screen "Lavados_Actuales" 1366x768, template "Pulsadores"
   Button "Botón_1" at 11,49 size 65x65; TextOff '1'
      on Click: SetTag("Ver_Anim_Boton", 1); SetTag("Ver_IDList", 0); "S400_ActListLav"(1)
      Appearance <- "Ver_Anim_Boton"
   IOField "Campo ES_1" at 115,75 size 95x32; FormatPattern 9999999999999999999999999999999999999999
      ProcessValue <- "Ver_HoraInicio_0"
   IOField "Campo ES_2" at 212,75 size 95x32; FormatPattern 9999999999999999999999999999999999999999
      ProcessValue <- "Ver_HoraFin_0"
   IOField "Campo ES_3" at 711,75 size 95x32; FormatPattern 99999
      ProcessValue <- "Ver_Carga_0"
   IOField "Campo ES_4" at 808,75 size 95x32; FormatPattern 99
      ProcessValue <- "Ver_Programa_0"
   IOField "Campo ES_5" at 309,75 size 400x32; FormatPattern ????????????????????????????????????????????????????????????????
      ProcessValue <- "Ver_Cli_Str_0"
   IOField "Campo ES_6" at 905,75 size 192x32; FormatPattern ????????????????????????????????????????????????????????????????
      ProcessValue <- "Ver_Operador_Str_0"
   IOField "Campo ES_7" at 115,106 size 95x32; FormatPattern 9999999999999999999999999999999999999999
      ProcessValue <- "Ver_HoraInicio_1"
   IOField "Campo ES_8" at 212,106 size 95x32; FormatPattern 9999999999999999999999999999999999999999
      ProcessValue <- "Ver_HoraFin_1"
   IOField "Campo ES_9" at 711,106 size 95x32; FormatPattern 99999
      ProcessValue <- "Ver_Carga_1"
   IOField "Campo ES_10" at 808,106 size 95x32; FormatPattern 99
      ProcessValue <- "Ver_Programa_1"
   IOField "Campo ES_11" at 309,106 size 400x32; FormatPattern ????????????????????????????????????????????????????????????????
      ProcessValue <- "Ver_Cli_Str_1"
   IOField "Campo ES_12" at 905,106 size 192x32; FormatPattern ????????????????????????????????????????????????????????????????
      ProcessValue <- "Ver_Operador_Str_1"
   IOField "Campo ES_13" at 115,137 size 95x32; FormatPattern 9999999999999999999999999999999999999999
      ProcessValue <- "Ver_HoraInicio_2"
   IOField "Campo ES_14" at 212,137 size 95x32; FormatPattern 9999999999999999999999999999999999999999
      ProcessValue <- "Ver_HoraFin_2"
   IOField "Campo ES_15" at 711,137 size 95x32; FormatPattern 99999
      ProcessValue <- "Ver_Carga_2"
   IOField "Campo ES_16" at 808,137 size 95x32; FormatPattern 99
      ProcessValue <- "Ver_Programa_2"
   IOField "Campo ES_17" at 309,137 size 400x32; FormatPattern ????????????????????????????????????????????????????????????????
      ProcessValue <- "Ver_Cli_Str_2"
   IOField "Campo ES_18" at 905,137 size 192x32; FormatPattern ????????????????????????????????????????????????????????????????
      ProcessValue <- "Ver_Operador_Str_2"
   IOField "Campo ES_19" at 115,168 size 95x32; FormatPattern 9999999999999999999999999999999999999999
      ProcessValue <- "Ver_HoraInicio_3"
   IOField "Campo ES_20" at 212,168 size 95x32; FormatPattern 9999999999999999999999999999999999999999
      ProcessValue <- "Ver_HoraFin_3"
   IOField "Campo ES_21" at 711,168 size 95x32; FormatPattern 99999
      ProcessValue <- "Ver_Carga_3"
   IOField "Campo ES_22" at 808,168 size 95x32; FormatPattern 99
      ProcessValue <- "Ver_Programa_3"
   IOField "Campo ES_23" at 309,168 size 400x32; FormatPattern ????????????????????????????????????????????????????????????????
      ProcessValue <- "Ver_Cli_Str_3"
   IOField "Campo ES_24" at 905,168 size 192x32; FormatPattern ????????????????????????????????????????????????????????????????
      ProcessValue <- "Ver_Operador_Str_3"
   IOField "Campo ES_25" at 115,199 size 95x32; FormatPattern 9999999999999999999999999999999999999999
      ProcessValue <- "Ver_HoraInicio_4"
   IOField "Campo ES_26" at 212,199 size 95x32; FormatPattern 9999999999999999999999999999999999999999
      ProcessValue <- "Ver_HoraFin_4"
   IOField "Campo ES_27" at 711,199 size 95x32; FormatPattern 99999
      ProcessValue <- "Ver_Carga_4"
   IOField "Campo ES_28" at 808,199 size 95x32; FormatPattern 99
      ProcessValue <- "Ver_Programa_4"
   IOField "Campo ES_29" at 309,199 size 400x32; FormatPattern ????????????????????????????????????????????????????????????????
      ProcessValue <- "Ver_Cli_Str_4"
   IOField "Campo ES_30" at 905,199 size 192x32; FormatPattern ????????????????????????????????????????????????????????????????
      ProcessValue <- "Ver_Operador_Str_4"
   IOField "Campo ES_31" at 115,230 size 95x32; FormatPattern 9999999999999999999999999999999999999999
      ProcessValue <- "Ver_HoraInicio_5"
   IOField "Campo ES_32" at 212,230 size 95x32; FormatPattern 9999999999999999999999999999999999999999
      ProcessValue <- "Ver_HoraFin_5"
   IOField "Campo ES_33" at 711,230 size 95x32; FormatPattern 99999
      ProcessValue <- "Ver_Carga_5"
   IOField "Campo ES_34" at 808,230 size 95x32; FormatPattern 99
      ProcessValue <- "Ver_Programa_5"
   IOField "Campo ES_35" at 309,230 size 400x32; FormatPattern ????????????????????????????????????????????????????????????????
      ProcessValue <- "Ver_Cli_Str_5"
   IOField "Campo ES_36" at 905,230 size 192x32; FormatPattern ????????????????????????????????????????????????????????????????
      ProcessValue <- "Ver_Operador_Str_5"
   IOField "Campo ES_37" at 115,261 size 95x32; FormatPattern 9999999999999999999999999999999999999999
      ProcessValue <- "Ver_HoraInicio_6"
   IOField "Campo ES_38" at 212,261 size 95x32; FormatPattern 9999999999999999999999999999999999999999
      ProcessValue <- "Ver_HoraFin_6"
   IOField "Campo ES_39" at 711,261 size 95x32; FormatPattern 99999
      ProcessValue <- "Ver_Carga_6"
   IOField "Campo ES_40" at 808,261 size 95x32; FormatPattern 99
      ProcessValue <- "Ver_Programa_6"
   IOField "Campo ES_41" at 309,261 size 400x32; FormatPattern ????????????????????????????????????????????????????????????????
      ProcessValue <- "Ver_Cli_Str_6"
   IOField "Campo ES_42" at 905,261 size 192x32; FormatPattern ????????????????????????????????????????????????????????????????
      ProcessValue <- "Ver_Operador_Str_6"
   IOField "Campo ES_43" at 115,292 size 95x32; FormatPattern 9999999999999999999999999999999999999999
      ProcessValue <- "Ver_HoraInicio_7"
   IOField "Campo ES_44" at 212,292 size 95x32; FormatPattern 9999999999999999999999999999999999999999
      ProcessValue <- "Ver_HoraFin_7"
   IOField "Campo ES_45" at 711,292 size 95x32; FormatPattern 99999
      ProcessValue <- "Ver_Carga_7"
   IOField "Campo ES_46" at 808,292 size 95x32; FormatPattern 99
      ProcessValue <- "Ver_Programa_7"
   IOField "Campo ES_47" at 309,292 size 400x32; FormatPattern ????????????????????????????????????????????????????????????????
      ProcessValue <- "Ver_Cli_Str_7"
   IOField "Campo ES_48" at 905,292 size 192x32; FormatPattern ????????????????????????????????????????????????????????????????
      ProcessValue <- "Ver_Operador_Str_7"
   IOField "Campo ES_49" at 115,323 size 95x32; FormatPattern 9999999999999999999999999999999999999999
      ProcessValue <- "Ver_HoraInicio_8"
   IOField "Campo ES_50" at 212,323 size 95x32; FormatPattern 9999999999999999999999999999999999999999
      ProcessValue <- "Ver_HoraFin_8"
   IOField "Campo ES_51" at 711,323 size 95x32; FormatPattern 99999
      ProcessValue <- "Ver_Carga_8"
   IOField "Campo ES_52" at 808,323 size 95x32; FormatPattern 99
      ProcessValue <- "Ver_Programa_8"
   IOField "Campo ES_53" at 309,323 size 400x32; FormatPattern ????????????????????????????????????????????????????????????????
      ProcessValue <- "Ver_Cli_Str_8"
   IOField "Campo ES_54" at 905,323 size 192x32; FormatPattern ????????????????????????????????????????????????????????????????
      ProcessValue <- "Ver_Operador_Str_8"
   IOField "Campo ES_55" at 115,354 size 95x32; FormatPattern 9999999999999999999999999999999999999999
      ProcessValue <- "Ver_HoraInicio_9"
   IOField "Campo ES_56" at 212,354 size 95x32; FormatPattern 9999999999999999999999999999999999999999
      ProcessValue <- "Ver_HoraFin_9"
   IOField "Campo ES_57" at 711,354 size 95x32; FormatPattern 99999
      ProcessValue <- "Ver_Carga_9"
   IOField "Campo ES_58" at 808,354 size 95x32; FormatPattern 99
      ProcessValue <- "Ver_Programa_9"
   IOField "Campo ES_59" at 309,354 size 400x32; FormatPattern ????????????????????????????????????????????????????????????????
      ProcessValue <- "Ver_Cli_Str_9"
   IOField "Campo ES_60" at 905,354 size 192x32; FormatPattern ????????????????????????????????????????????????????????????????
      ProcessValue <- "Ver_Operador_Str_9"
   IOField "Campo ES_61" at 115,385 size 95x32; FormatPattern 9999999999999999999999999999999999999999
      ProcessValue <- "Ver_HoraInicio_10"
   IOField "Campo ES_62" at 212,385 size 95x32; FormatPattern 9999999999999999999999999999999999999999
      ProcessValue <- "Ver_HoraFin_10"
   IOField "Campo ES_63" at 711,385 size 95x32; FormatPattern 99999
      ProcessValue <- "Ver_Carga_10"
   IOField "Campo ES_64" at 808,385 size 95x32; FormatPattern 99
      ProcessValue <- "Ver_Programa_10"
   IOField "Campo ES_65" at 309,385 size 400x32; FormatPattern ????????????????????????????????????????????????????????????????
      ProcessValue <- "Ver_Cli_Str_10"
   IOField "Campo ES_66" at 905,385 size 192x32; FormatPattern ????????????????????????????????????????????????????????????????
      ProcessValue <- "Ver_Operador_Str_10"
   IOField "Campo ES_67" at 115,416 size 95x32; FormatPattern 9999999999999999999999999999999999999999
      ProcessValue <- "Ver_HoraInicio_11"
   IOField "Campo ES_68" at 212,416 size 95x32; FormatPattern 9999999999999999999999999999999999999999
      ProcessValue <- "Ver_HoraFin_11"
   IOField "Campo ES_69" at 711,416 size 95x32; FormatPattern 99999
      ProcessValue <- "Ver_Carga_11"
   IOField "Campo ES_70" at 808,416 size 95x32; FormatPattern 99
      ProcessValue <- "Ver_Programa_11"
   IOField "Campo ES_71" at 309,416 size 400x32; FormatPattern ????????????????????????????????????????????????????????????????
      ProcessValue <- "Ver_Cli_Str_11"
   IOField "Campo ES_72" at 905,416 size 192x32; FormatPattern ????????????????????????????????????????????????????????????????
      ProcessValue <- "Ver_Operador_Str_11"
   IOField "Campo ES_73" at 115,447 size 95x32; FormatPattern 9999999999999999999999999999999999999999
      ProcessValue <- "Ver_HoraInicio_12"
   IOField "Campo ES_74" at 212,447 size 95x32; FormatPattern 9999999999999999999999999999999999999999
      ProcessValue <- "Ver_HoraFin_12"
   IOField "Campo ES_75" at 711,447 size 95x32; FormatPattern 99999
      ProcessValue <- "Ver_Carga_12"
   IOField "Campo ES_76" at 808,447 size 95x32; FormatPattern 99
      ProcessValue <- "Ver_Programa_12"
   IOField "Campo ES_77" at 309,447 size 400x32; FormatPattern ????????????????????????????????????????????????????????????????
      ProcessValue <- "Ver_Cli_Str_12"
   IOField "Campo ES_78" at 905,447 size 192x32; FormatPattern ????????????????????????????????????????????????????????????????
      ProcessValue <- "Ver_Operador_Str_12"
   IOField "Campo ES_79" at 115,478 size 95x32; FormatPattern 9999999999999999999999999999999999999999
      ProcessValue <- "Ver_HoraInicio_13"
   IOField "Campo ES_80" at 212,478 size 95x32; FormatPattern 9999999999999999999999999999999999999999
      ProcessValue <- "Ver_HoraFin_13"
   IOField "Campo ES_81" at 711,478 size 95x32; FormatPattern 99999
      ProcessValue <- "Ver_Carga_13"
   IOField "Campo ES_82" at 808,478 size 95x32; FormatPattern 99
      ProcessValue <- "Ver_Programa_13"
   IOField "Campo ES_83" at 309,478 size 400x32; FormatPattern ????????????????????????????????????????????????????????????????
      ProcessValue <- "Ver_Cli_Str_13"
   IOField "Campo ES_84" at 905,478 size 192x32; FormatPattern ????????????????????????????????????????????????????????????????
      ProcessValue <- "Ver_Operador_Str_13"
   IOField "Campo ES_85" at 115,509 size 95x32; FormatPattern 9999999999999999999999999999999999999999
      ProcessValue <- "Ver_HoraInicio_14"
   IOField "Campo ES_86" at 212,509 size 95x32; FormatPattern 9999999999999999999999999999999999999999
      ProcessValue <- "Ver_HoraFin_14"
   IOField "Campo ES_87" at 711,509 size 95x32; FormatPattern 99999
      ProcessValue <- "Ver_Carga_14"
   IOField "Campo ES_88" at 808,509 size 95x32; FormatPattern 99
      ProcessValue <- "Ver_Programa_14"
   IOField "Campo ES_89" at 309,509 size 400x32; FormatPattern ????????????????????????????????????????????????????????????????
      ProcessValue <- "Ver_Cli_Str_14"
   IOField "Campo ES_90" at 905,509 size 192x32; FormatPattern ????????????????????????????????????????????????????????????????
      ProcessValue <- "Ver_Operador_Str_14"
   TextField "Campo de texto_1" at 115,41 size 95x32; Text 'INICIO'
   TextField "Campo de texto_2" at 212,41 size 95x32; Text 'FIN'
   TextField "Campo de texto_3" at 309,41 size 95x32; Text 'CLIENTES'
   TextField "Campo de texto_4" at 711,41 size 95x32; Text 'CARGA'
   TextField "Campo de texto_5" at 808,41 size 95x32; Text 'PROG'
   TextField "Campo de texto_6" at 913,41 size 95x32; Text 'OPERADOR'
   Button "Botón_3" at 1145,665 size 39x38; TextOff 'Text'
      on Click: function_b9b71300("Ver_IDList", 1); "S400_ActListLav"("Ver_Anim_Boton")
   Button "Botón_4" at 1145,41 size 39x38; TextOff 'Text'
      on Click: function_dd21b452("Ver_IDList", 1); "S400_ActListLav"("Ver_Anim_Boton")
   Button "Botón_5" at 10,126 size 65x65; TextOff '2'
      on Click: SetTag("Ver_IDList", 0); SetTag("Ver_Anim_Boton", 2); "S400_ActListLav"(2)
      Appearance <- "Ver_Anim_Boton"
   Button "Botón_6" at 10,205 size 65x65; TextOff '3'
      on Click: SetTag("Ver_IDList", 0); SetTag("Ver_Anim_Boton", 3); "S400_ActListLav"(3)
      Appearance <- "Ver_Anim_Boton"
   Button "Botón_7" at 10,284 size 65x65; TextOff '4'
      on Click: SetTag("Ver_IDList", 0); SetTag("Ver_Anim_Boton", 4); "S400_ActListLav"(4)
      Appearance <- "Ver_Anim_Boton"
   IOField "Campo ES_91" at 115,541 size 95x32; FormatPattern 9999999999999999999999999999999999999999
      ProcessValue <- "Ver_HoraInicio_14"
   IOField "Campo ES_92" at 212,541 size 95x32; FormatPattern 9999999999999999999999999999999999999999
      ProcessValue <- "Ver_HoraFin_14"
   IOField "Campo ES_93" at 711,541 size 95x32; FormatPattern 99999
      ProcessValue <- "Ver_Carga_14"
   IOField "Campo ES_94" at 808,541 size 95x32; FormatPattern 99
      ProcessValue <- "Ver_Programa_14"
   IOField "Campo ES_95" at 309,541 size 400x32; FormatPattern ????????????????????????????????????????????????????????????????
      ProcessValue <- "Ver_Cli_Str_14"
   IOField "Campo ES_96" at 905,541 size 192x32; FormatPattern ????????????????????????????????????????????????????????????????
      ProcessValue <- "Ver_Operador_Str_14"
   IOField "Campo ES_97" at 115,573 size 95x32; FormatPattern 9999999999999999999999999999999999999999
      ProcessValue <- "Ver_HoraInicio_14"
   IOField "Campo ES_98" at 212,573 size 95x32; FormatPattern 9999999999999999999999999999999999999999
      ProcessValue <- "Ver_HoraFin_14"
   IOField "Campo ES_99" at 711,573 size 95x32; FormatPattern 99999
      ProcessValue <- "Ver_Carga_14"
   IOField "Campo ES_100" at 808,573 size 95x32; FormatPattern 99
      ProcessValue <- "Ver_Programa_14"
   IOField "Campo ES_101" at 309,573 size 400x32; FormatPattern ????????????????????????????????????????????????????????????????
      ProcessValue <- "Ver_Cli_Str_14"
   IOField "Campo ES_102" at 905,573 size 192x32; FormatPattern ????????????????????????????????????????????????????????????????
      ProcessValue <- "Ver_Operador_Str_14"
   IOField "Campo ES_103" at 115,605 size 95x32; FormatPattern 9999999999999999999999999999999999999999
      ProcessValue <- "Ver_HoraInicio_14"
   IOField "Campo ES_104" at 212,605 size 95x32; FormatPattern 9999999999999999999999999999999999999999
      ProcessValue <- "Ver_HoraFin_14"
   IOField "Campo ES_105" at 711,605 size 95x32; FormatPattern 99999
      ProcessValue <- "Ver_Carga_14"
   IOField "Campo ES_106" at 808,605 size 95x32; FormatPattern 99
      ProcessValue <- "Ver_Programa_14"
   IOField "Campo ES_107" at 309,605 size 400x32; FormatPattern ????????????????????????????????????????????????????????????????
      ProcessValue <- "Ver_Cli_Str_14"
   IOField "Campo ES_108" at 905,605 size 192x32; FormatPattern ????????????????????????????????????????????????????????????????
      ProcessValue <- "Ver_Operador_Str_14"
   IOField "Campo ES_109" at 115,637 size 95x32; FormatPattern 9999999999999999999999999999999999999999
      ProcessValue <- "Ver_HoraInicio_14"
   IOField "Campo ES_110" at 212,637 size 95x32; FormatPattern 9999999999999999999999999999999999999999
      ProcessValue <- "Ver_HoraFin_14"
   IOField "Campo ES_111" at 711,637 size 95x32; FormatPattern 99999
      ProcessValue <- "Ver_Carga_14"
   IOField "Campo ES_112" at 808,637 size 95x32; FormatPattern 99
      ProcessValue <- "Ver_Programa_14"
   IOField "Campo ES_113" at 309,637 size 400x32; FormatPattern ????????????????????????????????????????????????????????????????
      ProcessValue <- "Ver_Cli_Str_14"
   IOField "Campo ES_114" at 905,637 size 192x32; FormatPattern ????????????????????????????????????????????????????????????????
      ProcessValue <- "Ver_Operador_Str_14"
   IOField "Campo ES_115" at 115,669 size 95x32; FormatPattern 9999999999999999999999999999999999999999
      ProcessValue <- "Ver_HoraInicio_14"
   IOField "Campo ES_116" at 212,669 size 95x32; FormatPattern 9999999999999999999999999999999999999999
      ProcessValue <- "Ver_HoraFin_14"
   IOField "Campo ES_117" at 711,669 size 95x32; FormatPattern 99999
      ProcessValue <- "Ver_Carga_14"
   IOField "Campo ES_118" at 808,669 size 95x32; FormatPattern 99
      ProcessValue <- "Ver_Programa_14"
   IOField "Campo ES_119" at 309,669 size 400x32; FormatPattern ????????????????????????????????????????????????????????????????
      ProcessValue <- "Ver_Cli_Str_14"
   IOField "Campo ES_120" at 905,669 size 192x32; FormatPattern ????????????????????????????????????????????????????????????????
      ProcessValue <- "Ver_Operador_Str_14"
   TextField "Campo de texto_7" at 1099,75 size 32x32; Text 'X'
   TextField "Campo de texto_8" at 1099,106 size 32x32; Text 'X'
   TextField "Campo de texto_9" at 1099,137 size 32x32; Text 'X'
   TextField "Campo de texto_10" at 1099,168 size 32x32; Text 'X'
   TextField "Campo de texto_11" at 1099,199 size 32x32; Text 'X'
   TextField "Campo de texto_12" at 1099,230 size 32x32; Text 'X'
   TextField "Campo de texto_13" at 1099,261 size 32x32; Text 'X'
   TextField "Campo de texto_14" at 1099,292 size 32x32; Text 'X'
   TextField "Campo de texto_15" at 1099,323 size 32x32; Text 'X'
   TextField "Campo de texto_16" at 1099,354 size 32x32; Text 'X'
   TextField "Campo de texto_17" at 1099,385 size 32x32; Text 'X'
   TextField "Campo de texto_18" at 1099,416 size 32x32; Text 'X'
   TextField "Campo de texto_19" at 1099,447 size 32x32; Text 'X'
   TextField "Campo de texto_20" at 1099,478 size 32x32; Text 'X'
   TextField "Campo de texto_21" at 1099,509 size 32x32; Text 'X'
   TextField "Campo de texto_22" at 1099,541 size 32x32; Text 'X'
   TextField "Campo de texto_23" at 1099,573 size 32x32; Text 'X'
   TextField "Campo de texto_24" at 1099,605 size 32x32; Text 'X'
   TextField "Campo de texto_25" at 1099,637 size 32x32; Text 'X'
   TextField "Campo de texto_26" at 1099,669 size 32x32; Text 'X'
   Group "Group" at 1099,75 size 32x32
   Group "Group_1" at 1099,106 size 32x32
   Group "Group_2" at 1099,137 size 32x32
   Group "Group_3" at 1099,168 size 32x32
   Group "Group_4" at 1099,199 size 32x32
   Group "Group_5" at 1099,230 size 32x32
   Group "Group_6" at 1099,261 size 32x32
   Group "Group_7" at 1099,292 size 32x32
   Group "Group_8" at 1099,323 size 32x32
   Group "Group_9" at 1099,354 size 32x32
   Group "Group_10" at 1099,385 size 32x32
   Group "Group_11" at 1099,416 size 32x32
   Group "Group_12" at 1099,447 size 32x32
   Group "Group_13" at 1099,478 size 32x32
   Group "Group_14" at 1099,509 size 32x32
   Group "Group_15" at 1099,541 size 32x32
   Group "Group_16" at 1099,573 size 32x32
   Group "Group_17" at 1099,605 size 32x32
   Group "Group_18" at 1099,637 size 32x32
   Group "Group_19" at 1099,669 size 32x32
   Button "Botón_8" at 1200,75 size 32x32; TextOff 'E'
      Visibility <- "Ver_Programa_0"
      on Click: SetBit("Ver_Editor_X"); "S402_ActRegDeEdicion"("Ver_Anim_Boton", 0)
   Button "Botón_11" at 13,6 size 65x32; TextOff 'HOY'
      on Click: "S403_ActDia"()
   IOField "Campo ES_133" at 101,6 size 115x32; FormatPattern 9999999999999999999999999999999999999999
      ProcessValue <- "Ver_DIA_X"
   Button "Botón_13" at 1200,106 size 32x32; TextOff 'E'
      on Click: SetBit("Ver_Editor_X"); "S402_ActRegDeEdicion"("Ver_Anim_Boton", 1)
      Visibility <- "Ver_Programa_1"
   Button "Botón_14" at 1200,137 size 32x32; TextOff 'E'
      on Click: SetBit("Ver_Editor_X"); "S402_ActRegDeEdicion"("Ver_Anim_Boton", 2)
      Visibility <- "Ver_Programa_2"
   Button "Botón_15" at 1200,168 size 32x32; TextOff 'E'
      on Click: SetBit("Ver_Editor_X"); "S402_ActRegDeEdicion"("Ver_Anim_Boton", 3)
      Visibility <- "Ver_Programa_3"
   Button "Botón_16" at 1200,199 size 32x32; TextOff 'E'
      on Click: SetBit("Ver_Editor_X"); "S402_ActRegDeEdicion"("Ver_Anim_Boton", 4)
      Visibility <- "Ver_Programa_4"
   Button "Botón_17" at 1200,230 size 32x32; TextOff 'E'
      on Click: SetBit("Ver_Editor_X"); "S402_ActRegDeEdicion"("Ver_Anim_Boton", 5)
      Visibility <- "Ver_Programa_5"
   Button "Botón_18" at 1200,261 size 32x32; TextOff 'E'
      on Click: SetBit("Ver_Editor_X"); "S402_ActRegDeEdicion"("Ver_Anim_Boton", 6)
      Visibility <- "Ver_Programa_6"
   Button "Botón_19" at 1200,292 size 32x32; TextOff 'E'
      on Click: SetBit("Ver_Editor_X"); "S402_ActRegDeEdicion"("Ver_Anim_Boton", 7)
      Visibility <- "Ver_Programa_7"
   Button "Botón_20" at 1200,323 size 32x32; TextOff 'E'
      on Click: SetBit("Ver_Editor_X"); "S402_ActRegDeEdicion"("Ver_Anim_Boton", 8)
      Visibility <- "Ver_Programa_8"
   Button "Botón_21" at 1200,354 size 32x32; TextOff 'E'
      on Click: SetBit("Ver_Editor_X"); "S402_ActRegDeEdicion"("Ver_Anim_Boton", 9)
      Visibility <- "Ver_Programa_9"
   Button "Botón_22" at 1200,385 size 32x32; TextOff 'E'
      on Click: SetBit("Ver_Editor_X"); "S402_ActRegDeEdicion"("Ver_Anim_Boton", 10)
      Visibility <- "Ver_Programa_10"
   Button "Botón_23" at 1200,416 size 32x32; TextOff 'E'
      on Click: SetBit("Ver_Editor_X"); "S402_ActRegDeEdicion"("Ver_Anim_Boton", 11)
      Visibility <- "Ver_Programa_11"
   Button "Botón_24" at 1200,447 size 32x32; TextOff 'E'
      on Click: SetBit("Ver_Editor_X"); "S402_ActRegDeEdicion"("Ver_Anim_Boton", 12)
      Visibility <- "Ver_Programa_12"
   Button "Botón_25" at 1200,478 size 32x32; TextOff 'E'
      on Click: SetBit("Ver_Editor_X"); "S402_ActRegDeEdicion"("Ver_Anim_Boton", 13)
      Visibility <- "Ver_Programa_13"
   Button "Botón_26" at 1200,509 size 32x32; TextOff 'E'
      on Click: SetBit("Ver_Editor_X"); "S402_ActRegDeEdicion"("Ver_Anim_Boton", 14)
      Visibility <- "Ver_Programa_14"
   Button "Botón_27" at 1200,541 size 32x32; TextOff 'E'
      on Click: SetBit("Ver_Editor_X"); "S402_ActRegDeEdicion"("Ver_Anim_Boton", 15)
      Visibility <- "Ver_Programa_15"
   Button "Botón_29" at 1200,573 size 32x32; TextOff 'E'
      on Click: SetBit("Ver_Editor_X"); "S402_ActRegDeEdicion"("Ver_Anim_Boton", 16)
      Visibility <- "Ver_Programa_16"
   Button "Botón_30" at 1200,605 size 32x32; TextOff 'E'
      on Click: SetBit("Ver_Editor_X"); "S402_ActRegDeEdicion"("Ver_Anim_Boton", 17)
      Visibility <- "Ver_Programa_17"
   Button "Botón_31" at 1200,637 size 32x32; TextOff 'E'
      on Click: SetBit("Ver_Editor_X"); "S402_ActRegDeEdicion"("Ver_Anim_Boton", 18)
      Visibility <- "Ver_Programa_18"
   Button "Botón_32" at 1200,669 size 32x32; TextOff 'E'
      on Click: SetBit("Ver_Editor_X"); "S402_ActRegDeEdicion"("Ver_Anim_Boton", 19)
      Visibility <- "Ver_Programa_19"
   Button "Botón_2" at 1045,720 size 161x48; TextOff 'PRINCIPAL'
      on Click: ActivateScreen("Principal", 0)
   Button "Botón_12" at 405,720 size 161x48; TextOff 'GENERAR INFORME'
      on Click: "S23_Creador_InformeDiarioLavs_Gral"(N)
   Rectangle "Rectángulo_2" at 1099,75 size 32x32
      Visibility <- "Ver_CicloValido_0"
   Polygon "Polígono_3" at 1103,78 size 23x24
      Visibility <- "Ver_CicloValido_0"
   Rectangle "Rectángulo_3" at 1099,106 size 32x32
      Visibility <- "Ver_CicloValido_1"
   Polygon "Polígono_4" at 1103,109 size 23x24
      Visibility <- "Ver_CicloValido_1"
   Rectangle "Rectángulo_4" at 1099,137 size 32x32
      Visibility <- "Ver_CicloValido_2"
   Polygon "Polígono_5" at 1103,140 size 23x24
      Visibility <- "Ver_CicloValido_2"
   Rectangle "Rectángulo_5" at 1099,168 size 32x32
      Visibility <- "Ver_CicloValido_3"
   Polygon "Polígono_6" at 1103,171 size 23x24
      Visibility <- "Ver_CicloValido_3"
   Rectangle "Rectángulo_6" at 1099,199 size 32x32
      Visibility <- "Ver_CicloValido_4"
   Polygon "Polígono_7" at 1103,202 size 23x24
      Visibility <- "Ver_CicloValido_4"
   Rectangle "Rectángulo_7" at 1099,230 size 32x32
      Visibility <- "Ver_CicloValido_5"
   Polygon "Polígono_8" at 1103,233 size 23x24
      Visibility <- "Ver_CicloValido_5"
   Rectangle "Rectángulo_8" at 1099,261 size 32x32
      Visibility <- "Ver_CicloValido_6"
   Polygon "Polígono_9" at 1103,264 size 23x24
      Visibility <- "Ver_CicloValido_6"
   Rectangle "Rectángulo_9" at 1099,292 size 32x32
      Visibility <- "Ver_CicloValido_7"
   Polygon "Polígono_10" at 1103,295 size 23x24
      Visibility <- "Ver_CicloValido_7"
   Rectangle "Rectángulo_10" at 1099,323 size 32x32
      Visibility <- "Ver_CicloValido_8"
   Polygon "Polígono_11" at 1103,326 size 23x24
      Visibility <- "Ver_CicloValido_8"
   Rectangle "Rectángulo_11" at 1099,354 size 32x32
      Visibility <- "Ver_CicloValido_9"
   Polygon "Polígono_12" at 1103,357 size 23x24
      Visibility <- "Ver_CicloValido_9"
   Rectangle "Rectángulo_12" at 1099,385 size 32x32
      Visibility <- "Ver_CicloValido_10"
   Polygon "Polígono_13" at 1103,388 size 23x24
      Visibility <- "Ver_CicloValido_10"
   Rectangle "Rectángulo_13" at 1099,416 size 32x32
      Visibility <- "Ver_CicloValido_11"
   Polygon "Polígono_14" at 1103,419 size 23x24
      Visibility <- "Ver_CicloValido_11"
   Rectangle "Rectángulo_14" at 1099,447 size 32x32
      Visibility <- "Ver_CicloValido_12"
   Polygon "Polígono_15" at 1103,450 size 23x24
      Visibility <- "Ver_CicloValido_12"
   Rectangle "Rectángulo_15" at 1099,478 size 32x32
      Visibility <- "Ver_CicloValido_13"
   Polygon "Polígono_16" at 1103,481 size 23x24
      Visibility <- "Ver_CicloValido_13"
   Rectangle "Rectángulo_16" at 1099,509 size 32x32
      Visibility <- "Ver_CicloValido_14"
   Polygon "Polígono_17" at 1103,512 size 23x24
      Visibility <- "Ver_CicloValido_14"
   Rectangle "Rectángulo_17" at 1099,541 size 32x32
      Visibility <- "Ver_CicloValido_15"
   Polygon "Polígono_18" at 1103,544 size 23x24
      Visibility <- "Ver_CicloValido_15"
   Rectangle "Rectángulo_18" at 1099,573 size 32x32
      Visibility <- "Ver_CicloValido_16"
   Polygon "Polígono_19" at 1103,576 size 23x24
      Visibility <- "Ver_CicloValido_16"
   Rectangle "Rectángulo_19" at 1099,605 size 32x32
      Visibility <- "Ver_CicloValido_17"
   Polygon "Polígono_20" at 1103,608 size 23x24
      Visibility <- "Ver_CicloValido_17"
   Rectangle "Rectángulo_20" at 1099,637 size 32x32
      Visibility <- "Ver_CicloValido_18"
   Polygon "Polígono_21" at 1103,640 size 23x24
      Visibility <- "Ver_CicloValido_18"
   Rectangle "Rectángulo_21" at 1099,669 size 32x32
      Visibility <- "Ver_CicloValido_19"
   Polygon "Polígono_22" at 1103,672 size 23x24
      Visibility <- "Ver_CicloValido_19"
   Rectangle "Rectángulo_22" at 101,250 size 1086x267
      Visibility <- "Ver_Editor_X"
   TextField "Campo de texto_33" at 134,265 size 185x16; Text 'REGISTRO ACTUAL'
      Visibility <- "Ver_Editor_X"
   TextField "Campo de texto_27" at 115,289 size 95x16; Text 'INICIO'
      Visibility <- "Ver_Editor_X"
   TextField "Campo de texto_28" at 212,289 size 95x16; Text 'FIN'
      Visibility <- "Ver_Editor_X"
   IOField "Campo ES_122" at 212,311 size 95x32; FormatPattern 9999999999999999999999999999999999999999
      Visibility <- "Ver_Editor_X"
      ProcessValue <- "Ver_HoraFin_X_ans"
   IOField "Campo ES_121" at 115,311 size 95x32; FormatPattern 9999999999999999999999999999999999999999
      Visibility <- "Ver_Editor_X"
      ProcessValue <- "Ver_HoraInicio_X_ans"
   TextField "Campo de texto_29" at 309,289 size 95x16; Text 'CLIENTES'
      Visibility <- "Ver_Editor_X"
   IOField "Campo ES_123" at 711,311 size 95x32; FormatPattern 99999
      Visibility <- "Ver_Editor_X"
      ProcessValue <- "Ver_Carga_X_ans"
   TextField "Campo de texto_30" at 711,289 size 95x16; Text 'CARGA'
      Visibility <- "Ver_Editor_X"
   TextField "Campo de texto_31" at 808,289 size 95x16; Text 'PROG'
      Visibility <- "Ver_Editor_X"
   IOField "Campo ES_124" at 808,311 size 95x32; FormatPattern 99
      Visibility <- "Ver_Editor_X"
      ProcessValue <- "Ver_Programa_X_ans"
   TextField "Campo de texto_32" at 913,289 size 95x16; Text 'OPERADOR'
      Visibility <- "Ver_Editor_X"
   TextField "Campo de texto_39" at 913,388 size 95x16; Text 'OPERADOR'
      Visibility <- "Ver_Editor_X"
   TextField "Campo de texto_38" at 808,388 size 95x16; Text 'PROG'
      Visibility <- "Ver_Editor_X"
   TextField "Campo de texto_37" at 711,388 size 95x16; Text 'CARGA'
      Visibility <- "Ver_Editor_X"
   TextField "Campo de texto_35" at 212,388 size 95x16; Text 'FIN'
      Visibility <- "Ver_Editor_X"
   TextField "Campo de texto_40" at 134,364 size 185x16; Text 'REGISTRO NUEVO'
      Visibility <- "Ver_Editor_X"
   TextField "Campo de texto_34" at 115,388 size 95x16; Text 'INICIO'
      Visibility <- "Ver_Editor_X"
   Button "Botón_9" at 893,455 size 132x34; TextOff 'Guardar'
      Visibility <- "Ver_Editor_X"
      on Click: "S401_EditarLavado"("Ver_Anim_Boton"); ResetBit("Ver_Editor_X")
   Button "Botón_10" at 1035,455 size 132x34; TextOff 'Cancelar'
      Visibility <- "Ver_Editor_X"
      on Click: SetTag("Ver_CicloValido_X", 0); ResetBit("Ver_Editor_X")
   SymbolicIOField "Campo ES simbólico_2" at 309,407 size 400x32; TextOff '0'; TextOn '1'; TextList "Clientes"
      ProcessValue <- "Ver_Cli1_Str_X"
      Visibility <- "Ver_Editor_X"
   SymbolicIOField "Campo ES simbólico_1" at 309,441 size 400x32; TextOn '1'; TextOff '0'; TextList "Clientes"
      Visibility <- "Ver_Editor_X"
      ProcessValue <- "Ver_Cli2_Str_X"
   SymbolicIOField "Campo ES simbólico_3" at 309,475 size 400x32; TextOn '1'; TextOff '0'; TextList "Clientes"
      Visibility <- "Ver_Editor_X"
      ProcessValue <- "Ver_Cli3_Str_X"
   SymbolicIOField "Campo ES simbólico_4" at 905,407 size 192x32; TextOn '1'; TextOff '0'; TextList "Operadores_Lavadora"
      ProcessValue <- "Ver_Operador_Int_X"
      Visibility <- "Ver_Editor_X"
   IOField "Campo ES_131" at 808,407 size 95x32; FormatPattern 99
      ProcessValue <- "Ver_Programa_X"
      Visibility <- "Ver_Editor_X"
   IOField "Campo ES_129" at 711,407 size 95x32; FormatPattern 99999
      ProcessValue <- "Ver_Carga_X"
      Visibility <- "Ver_Editor_X"
   IOField "Campo ES_130" at 115,407 size 95x32; FormatPattern 9999999999999999999999999999999999999999
      ProcessValue <- "Ver_HoraInicio_X"
      Visibility <- "Ver_Editor_X"
   IOField "Campo ES_127" at 212,407 size 95x32; FormatPattern 9999999999999999999999999999999999999999
      ProcessValue <- "Ver_HoraFin_X"
      Visibility <- "Ver_Editor_X"
   SymbolicIOField "Campo ES simbólico_5" at 309,311 size 400x24; TextOn '1'; TextOff '0'; TextList "Clientes"
      Visibility <- "Ver_Editor_X"
      ProcessValue <- "Ver_Cli1_Str_X_ans"
   SymbolicIOField "Campo ES simbólico_6" at 309,337 size 400x24; TextOn '1'; TextOff '0'; TextList "Clientes"
      Visibility <- "Ver_Editor_X"
      ProcessValue <- "Ver_Cli2_Str_X_ans"
   SymbolicIOField "Campo ES simbólico_7" at 309,363 size 400x24; TextOn '1'; TextOff '0'; TextList "Clientes"
      Visibility <- "Ver_Editor_X"
      ProcessValue <- "Ver_Cli3_Str_X_ans"
   SymbolicIOField "Campo ES simbólico_8" at 905,311 size 192x32; TextOn '1'; TextOff '0'; TextList "Operadores_Lavadora"
      Visibility <- "Ver_Editor_X"
      ProcessValue <- "Ver_Operador_Int_X_ans"
   Switch "Interruptor_1" at 1099,311 size 63x32; CaptionText 'Switch'; TextOff 'NO'; TextOn 'SI'
      ProcessValue <- "Ver_CicloValido_X_ans"
      Visibility <- "Ver_Editor_X"
   Switch "Interruptor_2" at 1099,407 size 63x32; TextOn 'SI'; CaptionText 'Switch'; TextOff 'NO'
      ProcessValue <- "Ver_CicloValido_X"
      Visibility <- "Ver_Editor_X"

screen "Informes" 1366x768, template "Pulsadores"
   Button "Botón_3" at 725,720 size 161x48; TextOff 'LAVADOS'
      on Click: ActivateScreen("Lavados_Actuales", 0); "S403_ActDia"()
   Button "Botón_8" at 1045,720 size 161x48; TextOff 'PRINCIPAL'
      on Click: ActivateScreen("Principal", 0)
   Button "Botón_1" at 414,456 size 161x48; TextOff 'GENERAR INFORME'
      on Click: "S500_InformePeriodico"(1, "Inf_Ano", "Inf_Mes")
   IOField "Campo ES_1" at 167,456 size 50x48; FormatPattern 99
      ProcessValue <- "Inf_Mes"
   IOField "Campo ES_2" at 161,130 size 170x48; FormatPattern 9999999999999999999999999999999999999999
      ProcessValue <- "Inf_Desde"
   IOField "Campo ES_3" at 161,194 size 170x48; FormatPattern 9999999999999999999999999999999999999999
      ProcessValue <- "Inf_Hasta"
   TextField "Campo de texto_1" at 86,464 size 55x32; Text 'MES'
   TextField "Campo de texto_2" at 70,138 size 82x32; Text 'DESDE'
   TextField "Campo de texto_3" at 62,202 size 84x32; Text 'HASTA'
   Button "Botón_2" at 350,194 size 161x48; TextOff 'GENERAR INFORME'
      on Click: "S500_InformePeriodico"(0, "Inf_Desde", "Inf_Hasta")
   Button "Botón_4" at 254,594 size 161x48; TextOff 'GENERAR INFORME'
      on Click: "S500_InformePeriodico"(2, 0, "Inf_Ano")
   TextField "Campo de texto_4" at 94,408 size 238x32; Text 'INFORME MENSUAL'
   TextField "Campo de texto_5" at 94,88 size 260x32; Text 'INFORME PERIODICO'
   TextField "Campo de texto_6" at 94,552 size 204x32; Text 'INFORME ANUAL'
   IOField "Campo ES_4" at 150,594 size 84x48; FormatPattern 9999
      ProcessValue <- "Inf_Ano"
   TextField "Campo de texto_7" at 86,602 size 57x32; Text 'AÑO'
   IOField "Campo ES_5" at 310,456 size 84x48; FormatPattern 9999
      ProcessValue <- "Inf_Ano"
   TextField "Campo de texto_8" at 246,464 size 49x32; Text 'DEL'
   TextField "Campo de texto_9" at 278,42 size 149x32; Text 'LAVADORAS'
   TextField "Campo de texto_10" at 944,50 size 131x32; Text 'PLANCHAS'
   IOField "Campo ES_133" at 86,318 size 131x48; FormatPattern 9999999999999999999999999999999999999999
      ProcessValue <- "Ver_DIA_X"
   Button "Botón_12" at 230,318 size 161x48; TextOff 'GENERAR INFORME'
      on Click: "S23_Creador_InformeDiarioLavs_Gral"(N)
   TextField "Campo de texto_11" at 94,276 size 214x32; Text 'INFORME DIARIO'
   Button "Botón_6" at 1070,456 size 161x48; TextOff 'GENERAR INFORME'
      on Click: "S501_InformePer_Planchas"(1, "InfP_Ano", "InfP_Mes")
   IOField "Campo ES_6" at 823,456 size 50x48; FormatPattern 99
      ProcessValue <- "InfP_Mes"
   IOField "Campo ES_7" at 817,130 size 170x48; FormatPattern 9999999999999999999999999999999999999999
      ProcessValue <- "InfP_Desde"
   IOField "Campo ES_8" at 817,194 size 170x48; FormatPattern 9999999999999999999999999999999999999999
      ProcessValue <- "InfP_Hasta"
   TextField "Campo de texto_12" at 742,464 size 55x32; Text 'MES'
   TextField "Campo de texto_13" at 726,138 size 82x32; Text 'DESDE'
   TextField "Campo de texto_14" at 718,202 size 84x32; Text 'HASTA'
   Button "Botón_7" at 1006,194 size 161x48; TextOff 'GENERAR INFORME'
      on Click: "S501_InformePer_Planchas"(0, "InfP_Desde", "InfP_Hasta")
   Button "Botón_9" at 910,594 size 161x48; TextOff 'GENERAR INFORME'
      on Click: "S501_InformePer_Planchas"(2, 0, "InfP_Ano")
   TextField "Campo de texto_15" at 750,408 size 238x32; Text 'INFORME MENSUAL'
   TextField "Campo de texto_16" at 750,88 size 260x32; Text 'INFORME PERIODICO'
   TextField "Campo de texto_17" at 750,552 size 204x32; Text 'INFORME ANUAL'
   IOField "Campo ES_9" at 806,594 size 84x48; FormatPattern 9999
      ProcessValue <- "InfP_Ano"
   TextField "Campo de texto_18" at 742,602 size 57x32; Text 'AÑO'
   IOField "Campo ES_10" at 966,456 size 84x48; FormatPattern 9999
      ProcessValue <- "InfP_Ano"
   TextField "Campo de texto_19" at 902,464 size 49x32; Text 'DEL'
   IOField "Campo ES_11" at 742,318 size 131x48; FormatPattern 9999999999999999999999999999999999999999
      ProcessValue <- "Ver_DIA_XP"
   Button "Botón_10" at 886,318 size 161x48; TextOff 'GENERAR INFORME'
      on Click: "S07_InformeDiario_Planchas"(N)
   TextField "Campo de texto_20" at 750,276 size 214x32; Text 'INFORME DIARIO'

Template "Pulsadores" 1366x768
   Button "Botón_28" at 1205,720 size 161x48; TextOff 'Text'
   Button "Botón_2" at 1045,720 size 161x48; TextOff 'Text'
   Button "Botón_3" at 725,720 size 161x48; TextOff 'Text'
   Button "Botón_1" at 885,720 size 161x48; TextOff 'Text'
   Button "Botón_13" at 565,720 size 161x48; TextOff 'Text'
   Button "Botón_5" at 405,720 size 161x48; TextOff 'Text'

screen "TendenciasPL1_1" 1366x768, template "Pulsadores"
   TrendView "Visor de curvas_1" at 12,36 size 1338x326
   TrendView "Visor de curvas_2" at 12,394 size 1338x318
   TextField "Campo de texto_1" at 347,361 size 668x31; Text 'PRODUCTIVIDAD Y RENDIMIENTO CADA 15Min PLANCHA 1'
   TextField "Campo de texto_2" at 275,6 size 813x31; Text 'PRODUCTIVIDAD Y RENDIMIENTO ACUMULADO POR TURNO PLANCHA 1'
   Button "Botón_8" at 1045,720 size 161x48; TextOff 'PRINCIPAL'
      on Click: ActivateScreen("Principal", 0)

screen "Procesos" 1366x768
   TextField "Campo de texto_1" at 49,16 size 109x39; Text 'BRAUN'
   TextField "Campo de texto_2" at 49,80 size 103x23; Text 'ENJUAGUES'
   TextField "Campo de texto_3" at 49,112 size 90x23; Text 'INICIALES'
   TextField "Campo de texto_5" at 49,176 size 113x23; Text 'PRE-LAVADO'
   TextField "Campo de texto_10" at 49,336 size 88x23; Text 'LAVADO 1'
   TextField "Campo de texto_14" at 49,464 size 88x23; Text 'LAVADO 2'
   TextField "Campo de texto_18" at 49,592 size 103x23; Text 'ENJUAGUES'
   TextField "Campo de texto_19" at 49,624 size 74x23; Text 'FINALES'
   TextField "Campo de texto_20" at 49,656 size 137x23; Text 'CENTRIFUGADO'
   TextField "Campo de texto_27" at 193,80 size 94x23; Text 'CANTIDAD'
   TextField "Campo de texto_28" at 193,144 size 134x23; Text 'NIVEL DE AGUA'
   TextField "Campo de texto_29" at 193,112 size 70x23; Text 'TIEMPO'
   TextField "Campo de texto_30" at 193,208 size 134x23; Text 'NIVEL DE AGUA'
   TextField "Campo de texto_32" at 193,240 size 140x23; Text 'AGUA CALIENTE'
   TextField "Campo de texto_34" at 193,304 size 132x23; Text 'TEMPERATURA'
   TextField "Campo de texto_35" at 193,336 size 70x23; Text 'TIEMPO'
   TextField "Campo de texto_36" at 193,368 size 134x23; Text 'NIVEL DE AGUA'
   TextField "Campo de texto_37" at 193,400 size 140x23; Text 'AGUA CALIENTE'
   TextField "Campo de texto_38" at 193,432 size 132x23; Text 'TEMPERATURA'
   TextField "Campo de texto_39" at 193,464 size 70x23; Text 'TIEMPO'
   TextField "Campo de texto_40" at 193,496 size 134x23; Text 'NIVEL DE AGUA'
   TextField "Campo de texto_41" at 193,528 size 140x23; Text 'AGUA CALIENTE'
   TextField "Campo de texto_42" at 193,560 size 132x23; Text 'TEMPERATURA'
   TextField "Campo de texto_43" at 193,592 size 94x23; Text 'CANTIDAD'
   TextField "Campo de texto_44" at 193,624 size 70x23; Text 'TIEMPO'
   TextField "Campo de texto_45" at 193,656 size 70x23; Text 'TIEMPO'
   TextField "Campo de texto_4" at 193,272 size 63x23; Text 'VAPOR'
   TextField "Campo de texto_6" at 193,176 size 70x23; Text 'TIEMPO'
   IOField "Campo ES_1" at 394,656 size 80x24; FormatPattern FF; Unit  M
      ProcessValue <- "_Prog_Centr_Tiempo"
   IOField "Campo ES_2" at 394,592 size 80x24; FormatPattern F
      ProcessValue <- "_Prog_EnjFin_Cant"
   IOField "Campo ES_3" at 394,624 size 80x24; FormatPattern FF; Unit  M
      ProcessValue <- "_Prog_EnjFin_Tiempo"
   IOField "Campo ES_7" at 394,400 size 80x24; FormatPattern F
      ProcessValue <- "_Prog_Lav1_AgCaliente"
   IOField "Campo ES_8" at 394,368 size 80x24; FormatPattern F
      ProcessValue <- "_Prog_Lav1_NivAg"
   IOField "Campo ES_9" at 394,432 size 80x24; FormatPattern FF; Unit  °C
      ProcessValue <- "_Prog_Lav1_Temperatura"
   IOField "Campo ES_10" at 394,336 size 80x24; FormatPattern FF; Unit  M
      ProcessValue <- "_Prog_Lav1_Tiempo"
   IOField "Campo ES_11" at 394,528 size 80x24; FormatPattern F
      ProcessValue <- "_Prog_Lav2_AgCaliente"
   IOField "Campo ES_12" at 394,496 size 80x24; FormatPattern F
      ProcessValue <- "_Prog_Lav2_NivAg"
   IOField "Campo ES_13" at 394,560 size 80x24; FormatPattern FF; Unit °C
      ProcessValue <- "_Prog_Lav2_Temperatura"
   IOField "Campo ES_14" at 394,464 size 80x24; FormatPattern FF; Unit  M
      ProcessValue <- "_Prog_Lav2_Tiempo"
   IOField "Campo ES_15" at 394,240 size 80x24; FormatPattern F
      ProcessValue <- "_Prog_PreLav_AgCaliente"
   IOField "Campo ES_16" at 394,208 size 80x24; FormatPattern F
      ProcessValue <- "_Prog_PreLav_NivAg"
   IOField "Campo ES_17" at 394,304 size 80x24; FormatPattern FF; Unit  °C
      ProcessValue <- "_Prog_PreLav_Temperatura"
   IOField "Campo ES_18" at 394,176 size 80x24; FormatPattern FF; Unit  M
      ProcessValue <- "_Prog_PreLav_Tiempo"
   IOField "Campo ES_19" at 394,272 size 80x24; FormatPattern F
      ProcessValue <- "_Prog_PreLav_Vapor"
   IOField "Campo ES_4" at 394,80 size 80x24; FormatPattern F
      ProcessValue <- "_Prog_EnjIni_Cant"
   IOField "Campo ES_5" at 394,144 size 80x24; FormatPattern F
      ProcessValue <- "_Prog_EnjIni_NivAg"
   IOField "Campo ES_6" at 394,112 size 80x24; FormatPattern FF; Unit  M
      ProcessValue <- "_Prog_EnjIni_Tiempo"
   IOField "Campo ES_153" at 403,38 size 62x30; FormatPattern 99
      ProcessValue <- "_Prog_aModifBraun"
   Button "Botón_3" at 374,694 size 616x66; TextOff 'PRINCIPAL'
      on Click: ActivateScreen("Principal", 0)
   TextField "Campo de texto_7" at 280,42 size 102x23; Text 'PROGRAMA'
   Button "Botón_1" at 510,80 size 32x24; TextOff 'G'
      on Click: "S600_Cambiar_Vars_Todos"(1, 1)
   Button "Botón_2" at 510,112 size 32x24; TextOff 'G'
      on Click: "S600_Cambiar_Vars_Todos"(1, 2)
   Button "Botón_4" at 510,144 size 32x24; TextOff 'G'
      on Click: "S600_Cambiar_Vars_Todos"(1, 3)
   Button "Botón_5" at 510,176 size 32x24; TextOff 'G'
      on Click: "S600_Cambiar_Vars_Todos"(1, 4)
   Button "Botón_6" at 510,208 size 32x24; TextOff 'G'
      on Click: "S600_Cambiar_Vars_Todos"(1, 5)
   Button "Botón_7" at 510,240 size 32x24; TextOff 'G'
      on Click: "S600_Cambiar_Vars_Todos"(1, 6)
   Button "Botón_8" at 510,272 size 32x24; TextOff 'G'
      on Click: "S600_Cambiar_Vars_Todos"(1, 7)
   Button "Botón_9" at 510,304 size 32x24; TextOff 'G'
      on Click: "S600_Cambiar_Vars_Todos"(1, 8)
   Button "Botón_10" at 510,336 size 32x24; TextOff 'G'
      on Click: "S600_Cambiar_Vars_Todos"(1, 9)
   Button "Botón_11" at 510,368 size 32x24; TextOff 'G'
      on Click: "S600_Cambiar_Vars_Todos"(1, 10)
   Button "Botón_12" at 510,400 size 32x24; TextOff 'G'
      on Click: "S600_Cambiar_Vars_Todos"(1, 11)
   Button "Botón_13" at 510,432 size 32x24; TextOff 'G'
      on Click: "S600_Cambiar_Vars_Todos"(1, 12)
   Button "Botón_14" at 510,464 size 32x24; TextOff 'G'
      on Click: "S600_Cambiar_Vars_Todos"(1, 13)
   Button "Botón_15" at 510,496 size 32x24; TextOff 'G'
      on Click: "S600_Cambiar_Vars_Todos"(1, 14)
   Button "Botón_16" at 510,528 size 32x24; TextOff 'G'
      on Click: "S600_Cambiar_Vars_Todos"(1, 15)
   Button "Botón_17" at 510,560 size 32x24; TextOff 'G'
      on Click: "S600_Cambiar_Vars_Todos"(1, 16)
   Button "Botón_18" at 510,592 size 32x24; TextOff 'G'
      on Click: "S600_Cambiar_Vars_Todos"(1, 17)
   Button "Botón_19" at 510,624 size 32x24; TextOff 'G'
      on Click: "S600_Cambiar_Vars_Todos"(1, 18)
   Button "Botón_20" at 510,656 size 32x24; TextOff 'G'
      on Click: "S600_Cambiar_Vars_Todos"(1, 19)
   TextField "Campo de texto_8" at 713,24 size 123x39; Text 'GIRBAU'
   TextField "Campo de texto_9" at 713,88 size 103x23; Text 'ENJUAGUES'
   TextField "Campo de texto_11" at 713,120 size 90x23; Text 'INICIALES'
   TextField "Campo de texto_12" at 713,184 size 113x23; Text 'PRE-LAVADO'
   TextField "Campo de texto_13" at 713,344 size 88x23; Text 'LAVADO 1'
   TextField "Campo de texto_15" at 713,472 size 88x23; Text 'LAVADO 2'
   TextField "Campo de texto_16" at 713,600 size 103x23; Text 'ENJUAGUES'
   TextField "Campo de texto_17" at 713,632 size 74x23; Text 'FINALES'
   TextField "Campo de texto_21" at 713,664 size 137x23; Text 'CENTRIFUGADO'
   TextField "Campo de texto_22" at 857,88 size 94x23; Text 'CANTIDAD'
   TextField "Campo de texto_23" at 857,152 size 134x23; Text 'NIVEL DE AGUA'
   TextField "Campo de texto_24" at 857,120 size 70x23; Text 'TIEMPO'
   TextField "Campo de texto_25" at 857,216 size 134x23; Text 'NIVEL DE AGUA'
   TextField "Campo de texto_26" at 857,248 size 140x23; Text 'AGUA CALIENTE'
   TextField "Campo de texto_31" at 857,312 size 132x23; Text 'TEMPERATURA'
   TextField "Campo de texto_33" at 857,344 size 70x23; Text 'TIEMPO'
   TextField "Campo de texto_46" at 857,376 size 134x23; Text 'NIVEL DE AGUA'
   TextField "Campo de texto_47" at 857,408 size 140x23; Text 'AGUA CALIENTE'
   TextField "Campo de texto_48" at 857,440 size 132x23; Text 'TEMPERATURA'
   TextField "Campo de texto_49" at 857,472 size 70x23; Text 'TIEMPO'
   TextField "Campo de texto_50" at 857,504 size 134x23; Text 'NIVEL DE AGUA'
   TextField "Campo de texto_51" at 857,536 size 140x23; Text 'AGUA CALIENTE'
   TextField "Campo de texto_52" at 857,568 size 132x23; Text 'TEMPERATURA'
   TextField "Campo de texto_53" at 857,600 size 94x23; Text 'CANTIDAD'
   TextField "Campo de texto_54" at 857,632 size 70x23; Text 'TIEMPO'
   TextField "Campo de texto_55" at 857,664 size 70x23; Text 'TIEMPO'
   TextField "Campo de texto_56" at 857,280 size 63x23; Text 'VAPOR'
   TextField "Campo de texto_57" at 857,184 size 70x23; Text 'TIEMPO'
   IOField "Campo ES_20" at 1058,664 size 80x24; FormatPattern FF; Unit  M
      ProcessValue <- "_Prog_Centr_Tiempo"
   IOField "Campo ES_21" at 1058,600 size 80x24; FormatPattern F
      ProcessValue <- "_Prog_EnjFin_Cant"
   IOField "Campo ES_22" at 1058,632 size 80x24; FormatPattern FF; Unit  M
      ProcessValue <- "_Prog_EnjFin_Tiempo"
   IOField "Campo ES_23" at 1058,408 size 80x24; FormatPattern F
      ProcessValue <- "_Prog_Lav1_AgCaliente"
   IOField "Campo ES_24" at 1058,376 size 80x24; FormatPattern F
      ProcessValue <- "_Prog_Lav1_NivAg"
   IOField "Campo ES_25" at 1058,440 size 80x24; FormatPattern FF; Unit  °C
      ProcessValue <- "_Prog_Lav1_Temperatura"
   IOField "Campo ES_26" at 1058,344 size 80x24; FormatPattern FF; Unit  M
      ProcessValue <- "_Prog_Lav1_Tiempo"
   IOField "Campo ES_27" at 1058,536 size 80x24; FormatPattern F
      ProcessValue <- "_Prog_Lav2_AgCaliente"
   IOField "Campo ES_28" at 1058,504 size 80x24; FormatPattern F
      ProcessValue <- "_Prog_Lav2_NivAg"
   IOField "Campo ES_29" at 1058,568 size 80x24; FormatPattern FF; Unit °C
      ProcessValue <- "_Prog_Lav2_Temperatura"
   IOField "Campo ES_30" at 1058,472 size 80x24; FormatPattern FF; Unit  M
      ProcessValue <- "_Prog_Lav2_Tiempo"
   IOField "Campo ES_31" at 1058,248 size 80x24; FormatPattern F
      ProcessValue <- "_Prog_PreLav_AgCaliente"
   IOField "Campo ES_32" at 1058,216 size 80x24; FormatPattern F
      ProcessValue <- "_Prog_PreLav_NivAg"
   IOField "Campo ES_33" at 1058,312 size 80x24; FormatPattern FF; Unit  °C
      ProcessValue <- "_Prog_PreLav_Temperatura"
   IOField "Campo ES_34" at 1058,184 size 80x24; FormatPattern FF; Unit  M
      ProcessValue <- "_Prog_PreLav_Tiempo"
   IOField "Campo ES_35" at 1058,280 size 80x24; FormatPattern F
      ProcessValue <- "_Prog_PreLav_Vapor"
   IOField "Campo ES_36" at 1058,88 size 80x24; FormatPattern F
      ProcessValue <- "_Prog_EnjIni_Cant"
   IOField "Campo ES_37" at 1058,152 size 80x24; FormatPattern F
      ProcessValue <- "_Prog_EnjIni_NivAg"
   IOField "Campo ES_38" at 1058,120 size 80x24; FormatPattern FF; Unit  M
      ProcessValue <- "_Prog_EnjIni_Tiempo"
   IOField "Campo ES_39" at 1067,46 size 62x30; FormatPattern 99
      ProcessValue <- "_Prog_aModifGirbau"
   TextField "Campo de texto_58" at 944,50 size 102x23; Text 'PROGRAMA'
   Button "Botón_21" at 1174,88 size 32x24; TextOff 'G'
      on Click: "S600_Cambiar_Vars_Todos"(2, 1)
   Button "Botón_22" at 1174,120 size 32x24; TextOff 'G'
      on Click: "S600_Cambiar_Vars_Todos"(2, 2)
   Button "Botón_23" at 1174,152 size 32x24; TextOff 'G'
      on Click: "S600_Cambiar_Vars_Todos"(2, 3)
   Button "Botón_24" at 1174,184 size 32x24; TextOff 'G'
      on Click: "S600_Cambiar_Vars_Todos"(2, 4)
   Button "Botón_25" at 1174,216 size 32x24; TextOff 'G'
      on Click: "S600_Cambiar_Vars_Todos"(2, 5)
   Button "Botón_26" at 1174,248 size 32x24; TextOff 'G'
      on Click: "S600_Cambiar_Vars_Todos"(2, 6)
   Button "Botón_27" at 1174,280 size 32x24; TextOff 'G'
      on Click: "S600_Cambiar_Vars_Todos"(2, 7)
   Button "Botón_28" at 1174,312 size 32x24; TextOff 'G'
      on Click: "S600_Cambiar_Vars_Todos"(2, 8)
   Button "Botón_29" at 1174,344 size 32x24; TextOff 'G'
      on Click: "S600_Cambiar_Vars_Todos"(2, 9)
   Button "Botón_30" at 1174,376 size 32x24; TextOff 'G'
      on Click: "S600_Cambiar_Vars_Todos"(2, 10)
   Button "Botón_31" at 1174,408 size 32x24; TextOff 'G'
      on Click: "S600_Cambiar_Vars_Todos"(2, 11)
   Button "Botón_32" at 1174,440 size 32x24; TextOff 'G'
      on Click: "S600_Cambiar_Vars_Todos"(2, 12)
   Button "Botón_33" at 1174,472 size 32x24; TextOff 'G'
      on Click: "S600_Cambiar_Vars_Todos"(2, 13)
   Button "Botón_34" at 1174,504 size 32x24; TextOff 'G'
      on Click: "S600_Cambiar_Vars_Todos"(2, 14)
   Button "Botón_35" at 1174,536 size 32x24; TextOff 'G'
      on Click: "S600_Cambiar_Vars_Todos"(2, 15)
   Button "Botón_36" at 1174,568 size 32x24; TextOff 'G'
      on Click: "S600_Cambiar_Vars_Todos"(2, 16)
   Button "Botón_37" at 1174,600 size 32x24; TextOff 'G'
      on Click: "S600_Cambiar_Vars_Todos"(2, 17)
   Button "Botón_38" at 1174,632 size 32x24; TextOff 'G'
      on Click: "S600_Cambiar_Vars_Todos"(2, 18)
   Button "Botón_39" at 1174,664 size 32x24; TextOff 'G'
      on Click: "S600_Cambiar_Vars_Todos"(2, 19)
   Button "Botón_40" at 510,28 size 88x40; TextOff 'Actualizar Variables'
      on Click: "S601_Actualizar_Vars_Todos"(1)
   Button "Botón_41" at 1174,36 size 88x40; TextOff 'Actualizar Variables'
      on Click: "S601_Actualizar_Vars_Todos"(2)

VB script "S14_Write_data_Lav1"
   On Error Resume Next
   Dim hayError, K
   hayError = False
   
   If SmartTags("Lav1_GrabarBDD") = True Then
   
   	'Declaration of local tags
   	Dim conn, rst, SQL_Table
   	
   	Set conn = CreateObject("ADODB.Connection")
   	Set rst = CreateObject("ADODB.Recordset")
   	
   	'Abrir BBDD
   	conn.Open "Provider=MSDASQL;Initial Catalog=Lavadero;DSN=Lavadero"
   	
   	'Error routine
   	If Err.Number <> 0 Then
   		bfde4b54-0db7-4817-8032-87127bf19bb9 "Lav1: Error abrirb base #" & Err.Number & " " & Err.Description
   		hayError = True
   	End If
   		
   	' Recoleccion de datos de la lavadora 1 
   	Dim fechafin, fechainicio, cliente_0, cliente_1, cliente_2, operario, carga, programa, ciclovalido, falla, valido_CN
   	
   	
   	'fecha actual
   	fechafin = DateSerial(S12_Conversor_BCD_to_Int(SmartTags("Lav1_FchFin_Ano")), S12_Conversor_BCD_to_Int(SmartTags("Lav1_FchFin_Mes")), S12_Conversor_BCD_to_Int(SmartTags("Lav1_FchFin_Dia")))
   	fechafin = fechafin + TimeSerial(S12_Conversor_BCD_to_Int(SmartTags("Lav1_FchFin_Hr")), S12_Conversor_BCD_to_Int(SmartTags("Lav1_FchFin_Min")), S12_Conversor_BCD_to_Int(SmartTags("Lav1_FchFin_Seg")))
   	
   	'fecha de inicio del ciclo
   	fechainicio = DateSerial(S12_Conversor_BCD_to_Int(SmartTags("Lav1_FchIni_Ano")), S12_Conversor_BCD_to_Int(SmartTags("Lav1_FchIni_Mes")), S12_Conversor_BCD_to_Int(SmartTags("Lav1_FchIni_Dia")))
   	fechainicio = fechainicio + TimeSerial(S12_Conversor_BCD_to_Int(SmartTags("Lav1_FchIni_Hr")), S12_Conversor_BCD_to_Int(SmartTags("Lav1_FchIni_Min")), S12_Conversor_BCD_to_Int(SmartTags("Lav1_FchIni_Seg")))
   	
   	cliente_0 = SmartTags("Lav1_Cliente_0")
   	cliente_1 = SmartTags("Lav1_Cliente_1")
   	cliente_2 = SmartTags("Lav1_Cliente_2")
   		
   	operario = SmartTags("Lav1_Operador")
   	
   	carga = SmartTags("Lav1_CantRopa")
   	
   	programa =  S12_Conversor_BCD_to_Int(SmartTags("Lav1_Programa"))
   	
   	falla = SmartTags("Lav1_Falla")
   	
   	If SmartTags("Lav1_St_Ciclo") = 0 Then
   		valido_CN = 1
   	Else
   		valido_CN = 0
   	End If
   
   	If SmartTags("Lav1_St_Ciclo") = 0 Or  S12_Conversor_BCD_to_Int(SmartTags("Lav1_St_Ciclo")) > 13 Then	
   		ciclovalido = 1
   	Else
   		ciclovalido = 0
   	End If
   	
   	
   	'Definition of data record
   	SQL_Table = "INSERT INTO Lav1 VALUES ('"_
   		& fechafin & "' , '" _
   		& fechainicio & "' , '" _
   		& cliente_0 & "' , '" _
   		& cliente_1 & "' , '" _
   		& cliente_2 & "' , '" _
   		& operario & "' , '" _
   		& carga & "' , '" _
   		& programa & "' , '" _
   		& ciclovalido & "' , '" _
   		& valido_CN & "')"
   		
   	If hayError = False Then
   		'Execute
   		Set rst = conn.Execute(SQL_Table)
   	End If
   
   	' Se guarda en lavado anterior
   	SmartTags("Lav1_Programa_Anterior") = SmartTags("Lav1_Programa")
   	
   	'Error routine
   	If Err.Number <> 0 Then
   		bfde4b54-0db7-4817-8032-87127bf19bb9 "Error select Lav1: #" & Err.Number & " " & Err.Description
   		SmartTags("_errorNum1") = Err.Number
   		hayError = True
   	End If
   
   	If hayError = False Or SmartTags("Lav1_Cont_IntentosGrabado") >= 3 Then
   		'Tres confirmaciones diferentes si es que no se proceso la anterior, con loops se tilda
   		If SmartTags("Lav1_GrabarBDD") = True Then
   			SmartTags("Lav1_Ciclograbado") = True
   		End If
   		K = Timer + 2
   		Do While (Timer<K)
   		Loop
   		If SmartTags("Lav1_GrabarBDD") = True Then
   			SmartTags("Lav1_Ciclograbado") = True
   		End If
   	
   		
   		
   		If SmartTags("Lav1_Cont_IntentosGrabado") >= 3 Then
   			
   			'Envio email avisando que el ciclo no se grabo
   			cliente_0 = cliente_0 + cliente_1 + cliente_2
   			Call SA4_ErrorEnGrabBDD(1, fechafin, fechainicio, cliente_0,operario,carga,programa,ciclovalido)
   			
   			SmartTags("Lav1_Cont_IntentosGrabado") = 0
   			
   			If SmartTags("Lav1_GrabarBDD") = True Then
   				SmartTags("Lav1_Ciclograbado") = True
   			End If	
   		
   		End If
   		
   	Else
   			
   		SmartTags("Lav1_Cont_IntentosGrabado") = SmartTags("Lav1_Cont_IntentosGrabado") + 1
   	
   	End If
   
   End If
   
   
   ' Jump de error en esta linea
   	
   Err.Clear
   'Close data source 
   conn.close
   Set conn = Nothing
   Set rst = Nothing 
   	
   
   	

VB script "S12_Conversor_BCD_to_Int"
   '////////////////////////////////////////////////////////////////
   '		CONVERSOR DE BDC A UINT
   '////////////////////////////////////////////////////////////////
   
   
   Dim output, extracto
   'Parametros de subfuncion
   Dim BitMask, tmpMask, i, NewValue
   Dim pValue, pStartPos, pBits
   
   '////////////////////////////////////////////////////////////////
   '		Primeros 4 BITS
   
   '	Subfuncion
   	
   	pValue = Entrada
   	pStartPos = 4
   	pBits = 4
   
       For i = pStartPos - pBits + 1 To pStartPos
           If i < 32 Then 
   			tmpMask = 2 ^ (i - 1)
   		Else 
   			tmpMask = "&H80000000"
   		End If
           BitMask = BitMask Or tmpMask
       Next
       NewValue = CLng(pValue And BitMask)
   
       If NewValue And "&H80000000" Then 
   		tmpMask = pBits 
   	Else 
   		tmpMask = 0
   	End If
       NewValue = (NewValue And "&H7FFFFFFF") / 2 ^ (pStartPos - pBits)
       If tmpMask Then
           If tmpMask < 32 Then 
   			BitMask = 2 ^ (tmpMask - 1) 
   		Else 
   			BitMask = "&H80000000"
   		End If
           NewValue = NewValue Or BitMask
       End If
       extracto = CLng(NewValue)
   '	End subfuncion
   
   output = extracto
   
   '////////////////////////////////////////////////////////////////
   '		SEGUNDOS 4 BITS
   
   '	Subfuncion
   	pValue = Entrada
   	pStartPos = 8
   	pBits = 4
   	BitMask = 0
   
       For i = pStartPos - pBits + 1 To pStartPos
           If i < 32 Then 
   			tmpMask = 2 ^ (i - 1)
   		Else 
   			tmpMask = "&H80000000"
   		End If
           BitMask = BitMask Or tmpMask
       Next
       NewValue = CLng(pValue And BitMask)
       SmartTags("bitmask") = BitMask
       If NewValue And "&H80000000" Then 
   		tmpMask = pBits 
   	Else 
   		tmpMask = 0
   	End If
       NewValue = (NewValue And "&H7FFFFFFF") / 2 ^ (pStartPos - pBits)
       If tmpMask Then
           If tmpMask < 32 Then 
   			BitMask = 2 ^ (tmpMask - 1) 
   		Else 
   			BitMask = "&H80000000"
   		End If
           NewValue = NewValue Or BitMask
       End If
       extracto = CLng(NewValue)
   '	End subfuncion
   
   output = output + extracto *10
   
   '////////////////////////////////////////////////////////////////
   '		TERCEROS 4 BITS
   '	Subfuncion
   	pValue = Entrada
   	pStartPos = 12
   	pBits = 4
   	BitMask = 0
   
       For i = pStartPos - pBits + 1 To pStartPos
           If i < 32 Then 
   			tmpMask = 2 ^ (i - 1)
   		Else 
   			tmpMask = "&H80000000"
   		End If
           BitMask = BitMask Or tmpMask
       Next
       NewValue = CLng(pValue And BitMask)
       If NewValue And "&H80000000" Then 
   		tmpMask = pBits 
   	Else 
   		tmpMask = 0
   	End If
       NewValue = (NewValue And "&H7FFFFFFF") / 2 ^ (pStartPos - pBits)
       If tmpMask Then
           If tmpMask < 32 Then 
   			BitMask = 2 ^ (tmpMask - 1) 
   		Else 
   			BitMask = "&H80000000"
   		End If
           NewValue = NewValue Or BitMask
       End If
       extracto = CLng(NewValue)
   '	End subfuncion
   
   
   output = output + extracto *100
   
   '////////////////////////////////////////////////////////////////
   '		CUARTOS 4 BITS
   '	Subfuncion
   	pValue = Entrada
   	pStartPos = 16
   	pBits = 4
   	BitMask = 0
   	
       For i = pStartPos - pBits + 1 To pStartPos
           If i < 32 Then 
   			tmpMask = 2 ^ (i - 1)
   		Else 
   			tmpMask = "&H80000000"
   		End If
           BitMask = BitMask Or tmpMask
       Next
       NewValue = CLng(pValue And BitMask)
       If NewValue And "&H80000000" Then 
   		tmpMask = pBits 
   	Else 
   		tmpMask = 0
   	End If
       NewValue = (NewValue And "&H7FFFFFFF") / 2 ^ (pStartPos - pBits)
       If tmpMask Then
           If tmpMask < 32 Then 
   			BitMask = 2 ^ (tmpMask - 1) 
   		Else 
   			BitMask = "&H80000000"
   		End If
           NewValue = NewValue Or BitMask
       End If
       extracto = CLng(NewValue)
   '	End subfuncion
   
   output = output + extracto *1000
   
   
   'Salida
   S12_Conversor_BCD_to_Int = output

VB script "S07_InformeDiario_Planchas"
   S07_InformeDiario_Planchas = "ERROR"
   
   'Declaration of local tags - Deklaration von lokalem Variablen
   Dim conn, rst, SQL_Table, i, j, horarioTurno(4)
   
   Dim Consulta
   
   On Error Resume Next
   
   Set conn = CreateObject("ADODB.Connection")
   Set rst = CreateObject("ADODB.Recordset")
   
   'Open data source - Datenquelle öffnen
   conn.Open "Provider=MSDASQL;Initial Catalog=Lavadero;DSN=Lavadero"
   'Error routine - Fehlerroutine
   If Err.Number <> 0 Then
   	bfde4b54-0db7-4817-8032-87127bf19bb9 "Conexion Error #" & Err.Number & " " & Err.Description
   	Err.Clear
   	conn.close
   	Set conn = Nothing  
   	Exit Function
   End If
   
   ' #################   Generacion de consulta a BDD Plancha1   ######################
   
   Dim DiaAnterior
   DiaAnterior = SmartTags("Ver_DIA_XP")
   'DiaAnterior = DateAdd("d",-1, DiaAnterior)
   SmartTags("tmp_prueba_5") = DiaAnterior
   
   SmartTags("Inf_FechaInforme") 			= DiaAnterior
   SmartTags("Inf_FechaInforme_WeekDay") 	= Weekday(DiaAnterior)
   
   Consulta = "SELECT * FROM Plancha1 WHERE cast(Fecha As Date) = '"
   Consulta = Consulta & CStr(Year(DiaAnterior)) & "-" & CStr(Month(DiaAnterior)) & "-" & CStr(Day(DiaAnterior)) & "' "
   Consulta = Consulta & "order by Fecha"
   
   'Execute
   Set rst = conn.Execute(Consulta)
   
   'Error routine
   If Err.Number <> 0 Then
   	bfde4b54-0db7-4817-8032-87127bf19bb9 "Consulta1 PL1 Error #" & Err.Number & " " & Err.Description
   	Err.Clear
   	'Close data source - Datenquelle schließen0
   	conn.close
   	Set conn = Nothing
   	Set rst = Nothing 
   	Exit Function
   End If
   	
   '####################### PROCESAMIENTO DE DATOS PLANCHA 1 ########################
   
       Dim iTotal(5)
       Dim iProd(5)
       Dim iRend(5)
   	Dim iRendPesado(5)
   
       Dim Total(5)
       Dim Prod(5)
       Dim Rend(5)
       
       Dim personas(5)
       Dim indice(5)
       
       Dim RendPesado(5)
       
       Dim Tmp(5)
               
       Dim XProd(5)
       Dim XRend(5)
       Dim XRendPesado(5)
       
       Dim diasEnHorasT(5), diasEnHorasP(5), diasEnHorasR(5)
       
       '' Recoleccion de tiempos de la consulta
       
       For i = 1 To 5
   		personas(i) = 0
   	Next
   	
       
       j = 1
       For i = 1 To 5
   	    iTotal(i) 		= CDbl(rst.Fields(j).Value) / 100.0
   	    j = j + 1
   	    iProd(i) 		= CDbl(rst.Fields(j).Value) / 100.0
   	    j = j + 1
   	    iRend(i) 		= CDbl(rst.Fields(j).Value) / 100.0
   	    j = j + 2
       Next
   
   If Err.Number <> 0 Then
   	bfde4b54-0db7-4817-8032-87127bf19bb9 "Recoleccion de Datos PL1 Error #" & Err.Number & " " & Err.Description
   	Err.Clear
   	Exit Function
   End If
               
       rst.MoveNext
       
       Do While rst.EOF = False
           
           j = 1
           For i = 1 To 5
   	        Total(i) = CDbl(rst.Fields(j).Value) / 100.0
   	        j = j + 1
   	        Prod(i) = CDbl(rst.Fields(j).Value) / 100.0
   	        j = j + 1
   	        Rend(i) = CDbl(rst.Fields(j).Value) / 100.0
   	        j = j + 2
   	        'Cantidad de operadores
   	        
   	        If InStr(CStr(rst.Fields(61).Value), "V") Then
   	        	personas(2) = rst.Fields(75).Value
   			End If
   			
   			If InStr(CStr(rst.Fields(62).Value), "V") Then
   	        	personas(3) = rst.Fields(75).Value
   			End If
   						
   			If InStr(CStr(rst.Fields(63).Value), "V") Then
   	        	personas(4) = rst.Fields(75).Value
   			End If
   									
   		    If InStr(CStr(rst.Fields(64).Value), "V") Then
   	        	personas(5) = rst.Fields(75).Value
   			End If
   			
           Next
           
           rst.MoveNext
           
   	Loop  
   	
   	If Err.Number <> 0 Then
   		bfde4b54-0db7-4817-8032-87127bf19bb9 "Recoleccion de Datos2 PL1 Error #" & Err.Number & " " & Err.Description
   		Err.Clear
   		Exit Function
   	End If       
       
       'Calculo de tiempos totales
   
       For i = 1 To 5
           Total(i) 	= (Total(i) - iTotal(i)) 	/ 86400.0
           Prod(i) 	= (Prod(i) - iProd(i)) 		/ 86400.0
           Rend(i) 	= (Rend(i) - iRend(i)) 		/ 86400.0   
           'Incremento indice de bucle
   	Next
   	
     personas(1) = personas(2) + personas(3) + personas(4) + personas(5) 
     
   	If Err.Number <> 0 Then
   		bfde4b54-0db7-4817-8032-87127bf19bb9 "Procesamiento final Datos PL1 Error #" & Err.Number & " " & Err.Description
   		Err.Clear
   		Exit Function
   	End If
   
   conn.close
   Set rst = Nothing
   Set conn = Nothing
   
   ' #################   Generacion de consulta a BDD Plancha2   ######################
   
   Dim conn2, rst2
   Set conn2 = CreateObject("ADODB.Connection")
   Set rst2 = CreateObject("ADODB.Recordset")
   
   'Open data source - Datenquelle öffnen
   conn2.Open "Provider=MSDASQL;Initial Catalog=Lavadero;DSN=Lavadero"
   'Error routine - Fehlerroutine
   If Err.Number <> 0 Then
   	bfde4b54-0db7-4817-8032-87127bf19bb9 "Conexion2 Error #" & Err.Number & " " & Err.Description
   	Err.Clear
   	Set conn2 = Nothing  
   	Exit Function
   End If
   
   '## Consulta de planchadora2
   Consulta = "SELECT * FROM Plancha2 WHERE cast(Fecha As Date) = '"
   Consulta = Consulta & CStr(Year(DiaAnterior)) & "-" & CStr(Month(DiaAnterior)) & "-" & CStr(Day(DiaAnterior)) & "' "
   Consulta = Consulta & " order by Fecha"
   
   
   'Execute - Ausführen
   Set rst2 = conn2.Execute(Consulta)
   
   'Error routine - Fehler Routine
   If Err.Number <> 0 Then
   	bfde4b54-0db7-4817-8032-87127bf19bb9 "Consulta PL2 Error #" & Err.Number & " " & Err.Description
   	Err.Clear
   	'Close data source - Datenquelle schließen
   	conn2.close
   	Set conn2 = Nothing
   	Set rst2 = Nothing
   End If
   	
   '####################### PROCESAMIENTO DE DATOS PLANCHA 2 ########################
   
       Dim iTotal2(5)
       Dim iProd2(5)
       Dim iRend2(5)
   	Dim iRendPesado2(5)
   
       Dim Total2(5), strTotal2(5)
       Dim Prod2(5), strProd2(5)
       Dim Rend2(5), strRend2(5)
       
       Dim RendPesado2(5)
       
       Dim Tmp2(5)
               
       Dim XProd2(5)
       Dim XRend2(5)
       Dim XRendPesado2(5)
   
   
   ' Recoleccion de tiempos de la consulta
       
       j = 1
       For i = 1 To 5
   	    iTotal2(i) 		= CDbl(rst2.Fields(j).Value) / 100.0
   	    j = j + 1
   	    iProd2(i) 		= CDbl(rst2.Fields(j).Value) / 100.0
   	    j = j + 1
   	    iRend2(i) 		= CDbl(rst2.Fields(j).Value) / 100.0
   	    j = j + 2
   	Next
   	
   If Err.Number <> 0 Then
   	bfde4b54-0db7-4817-8032-87127bf19bb9 "Error, Extraccion en consulta por planchadora2 en primera linea, Error Nro:" & Err.Number & " : " & Err.Description
   	Err.Clear
   End If
               
       rst2.MoveNext
       
       Do While rst2.EOF = False
           
           j = 1
           For i = 1 To 5
   	        Total2(i) 	= CDbl(rst2.Fields(j).Value) / 100.0
   	        j = j + 1
   	        Prod2(i) 	= CDbl(rst2.Fields(j).Value) / 100.0
   	        j = j + 1
   	        Rend2(i) 	= CDbl(rst2.Fields(j).Value) / 100.0
   	        j = j + 2
           Next
           
           rst2.MoveNext
           
       Loop        
       
    If Err.Number <> 0 Then
   	bfde4b54-0db7-4817-8032-87127bf19bb9 "Error, Extraccion en consulta por planchadora2, Error Nro:" & Err.Number & " : " & Err.Description
   	Err.Clear
   End If
       
       'Calculo de tiempos totales
   Dim aux0(5),aux1(5),aux2(5)
   
       For i = 1 To 5
           aux0(i) = (Total2(i) - iTotal2(i)) / 86400.0
           aux1(i) = (Prod2(i) - iProd2(i)) / 86400.0
           aux2(i) = (Rend2(i) - iRend2(i)) / 86400.0
           
           Total2(i) 	= Total(i) + aux0(i)
           Prod2(i) 	= Prod(i) + aux1(i)
           Rend2(i) 	= Rend(i) + aux2(i)
           
           'Obtengo los porcentajes de tiempos
           
          	If Total2(i) <> 0 Then
               XProd2(i) = 100.0 * (Prod2(i) / Total2(i))
               XRend2(i) = 100.0 * (Rend2(i) / Total2(i))
           Else
               XProd2(i) = 0.0
               XRend2(i) = 0.0
   		End If
           
           'Incremento indice de bucle
   	Next
           
   'Error routine
   If Err.Number <> 0 Then
   	bfde4b54-0db7-4817-8032-87127bf19bb9 "Conexion Error Calculo de Porcentajes, Error Nro:" & Err.Number & " : " & Err.Description
   	Err.Clear
   End If
   
   ' Pasaje de diashoras  a horas
   		
   For i= 1 To 5
   	diasEnHorasT(i) = Fix(Total2(i)) / 1
   	Total2(i) 		= Total2(i) - diasEnHorasT(i)
   	strTotal2(i) 	= SA2_TotalTimeToString(diasEnHorasT(i), Total2(i))
   	
   	
   	diasEnHorasP(i) = Fix(Prod2(i)) / 1
   	Prod2(i) 		= Prod2(i) - diasEnHorasP(i)
   	strProd2(i) 	= SA2_TotalTimeToString(diasEnHorasP(i), Prod2(i))
   	
   	
   	diasEnHorasR(i) = Fix(Rend2(i)) / 1
   	Rend2(i) 		= Rend2(i) - diasEnHorasR(i)
   	strRend2(i) 	= SA2_TotalTimeToString(diasEnHorasR(i), Rend2(i))
   Next
   
   
   
   'Close data source - Datenquelle schließen
   
   conn2.close
   Set rst = Nothing
   Set conn2 = Nothing
   
   '///////////////////////////////     Extraccion de Indices   /////////////////
   Dim connindx, rstindx, Consultaindx, listaIndices(60), k
   
   Set connindx = CreateObject("ADODB.Connection")
   Set rstindx = CreateObject("ADODB.Recordset")
   
   'Open data source - Datenquelle öffnen
   connindx.Open "Provider=MSDASQL;Initial Catalog=Lavadero;DSN=Lavadero"
   'Error routine - Fehlerroutine
   If Err.Number <> 0 Then
   	bfde4b54-0db7-4817-8032-87127bf19bb9 "Conexion Error a indicesPlanchas" & Err.Number & " " & Err.Description
   	Err.Clear
   	Set connindx = Nothing  
   End If
   
   Consultaindx = "SELECT * FROM indicesPlanchas;"
   
   'Ejecutar consulta
   Set rstindx = connindx.Execute(Consultaindx)
   
   ' Establecer los indices
   j = 1
   k = 1
   Do While rstindx.EOF = False
   	For j = 1 To 5
   		If (rstindx.Fields(0).Value = personas(j)) Then ' Si el ciclo es no valido
   			indice(j) = rstindx.Fields(1).Value / 10.0
   		End If
   	Next
   	
   	'Para imprimir todos los indices
   	listaIndices(k) = rstindx.Fields(1).Value / 10.0
   	k = k + 1
   	
   	rstindx.MoveNext
   Loop
   
   If Err.Number <> 0 Then
   	bfde4b54-0db7-4817-8032-87127bf19bb9 "Error en establecer los operadores#" & Err.Number & " " & Err.Description
   	Err.Clear
   	Set connindx = Nothing  
   	Exit Function
   End If
   
   
   
   
   'Creo Excel
   Dim objExcel, fila
   
   fila = 5
   Set objExcel = CreateObject("Excel.Application")
   
   objExcel.Visible = False
   
   objExcel.Workbooks.Open "C:\ESPACIO DE TRABAJO\InformeDiario\Plantillas\InformeDiarioExcel.xlsx"
       
       ' Fecha informe
   	objExcel.Cells(2,5).Value 		= DiaAnterior
   
       'Plancha 1
       objExcel.Cells(fila,3).Value 		= strTotal2			(1)
       objExcel.Cells(fila,4).Value 		= strProd2 			(1)
       objExcel.Cells(fila,5).Value 		= XProd2 			(1)
   	objExcel.Cells(fila,6).Value 		= strRend2			(1)
   	objExcel.Cells(fila,7).Value 		= XRend2 			(1)
   	objExcel.Cells(fila,8).Value 		= personas 			(1)
   	objExcel.Cells(fila,9).Value 		= indice 			(1)
   	
   If Err.Number <> 0 Then
   	bfde4b54-0db7-4817-8032-87127bf19bb9 "Asignasion Datos PL1 Error #" & Err.Number & " " & Err.Description
   	Err.Clear 
   End If
   
   Dim tmp_hour_ini, tmp_hour_fin, tmp_01, min_01, str_min_01
   
   tmp_01 = CStr(SmartTags("Inf_FechaInforme_WeekDay"))
   
   
   
   For i = 1 To 3
   	horarioTurno(i) = CStr(Hour(SmartTags("Planchadora1_Supervisores{"& CStr(i) &"}_Diadelasemana{" & tmp_01 & "}_Entrda")))
   		min_01 = Minute(SmartTags("Planchadora1_Supervisores{"& CStr(i) &"}_Diadelasemana{" & tmp_01 & "}_Entrda"))
   		If min_01 < 10 Then
   			str_min_01 = "0" + CStr(min_01)
   		Else
   			str_min_01 = CStr(min_01)
   		End If
   	
   	horarioTurno(i) = horarioTurno(i) & ":" & str_min_01
   	horarioTurno(i) = horarioTurno(i) & "/" & CStr(Hour(SmartTags("Planchadora1_Supervisores{"& CStr(i) &"}_Diadelasemana{" & tmp_01 & "}_Salida")))
   	
   		min_01 = Minute(SmartTags("Planchadora1_Supervisores{"& CStr(i) &"}_Diadelasemana{" & tmp_01 & "}_Salida"))
   		If min_01 < 10 Then
   			str_min_01 = "0" + CStr(min_01)
   		Else
   			str_min_01 = CStr(min_01)
   		End If
   	
   	horarioTurno(i) = horarioTurno(i) & ":" & str_min_01
   Next
   
   	horarioTurno(4) = CStr(Hour(SmartTags("Planchadora1_Supervisores{4}_Diadelasemana{" & tmp_01 & "}_Entrada")))
   			min_01 = Minute(SmartTags("Planchadora1_Supervisores{4}_Diadelasemana{" & tmp_01 & "}_Entrda"))
   		If min_01 < 10 Then
   			str_min_01 = "0" + CStr(min_01)
   		Else
   			str_min_01 = CStr(min_01)
   		End If
   	horarioTurno(4) = horarioTurno(4) & ":" & min_01
   	horarioTurno(4) = horarioTurno(4) & "/" & CStr(Hour(SmartTags("Planchadora1_Supervisores{4}_Diadelasemana{" & tmp_01 & "}_Salida")))
   		min_01 = Minute(SmartTags("Planchadora1_Supervisores{4}_Diadelasemana{" & tmp_01 & "}_Salida"))
   		If min_01 < 10 Then
   			str_min_01 = "0" + CStr(min_01)
   		Else
   			str_min_01 = CStr(min_01)
   		End If
   	horarioTurno(4) = horarioTurno(4) & ":" & min_01
   
   	'Supervisores
   For i = 1 To 4 
   	
   	objExcel.Cells(i+fila,2).Value 		= horarioTurno		(i)
   	objExcel.Cells(i+fila,3).Value 		= strTotal2			(i+1)
   	objExcel.Cells(i+fila,4).Value 		= strProd2			(i+1)
   	objExcel.Cells(i+fila,5).Value 		= XProd2 			(i+1)
   	objExcel.Cells(i+fila,6).Value 		= strRend2			(i+1)
   	objExcel.Cells(i+fila,7).Value	    = XRend2			(i+1)
   	objExcel.Cells(i+fila,8).Value	    = personas			(i+1)
   	objExcel.Cells(i+fila,9).Value 		= indice 			(i+1)
   	
   	If Err.Number <> 0 Then
   		bfde4b54-0db7-4817-8032-87127bf19bb9 "Asignasion Datos Sup"& CStr(i) &" PL1 Error #" & Err.Number & " " & Err.Description
   		Err.Clear
   	End If
   Next
   
   For j = 1 To 4
   	If 0 = personas(j+1) Then ' Si el ciclo es no valido
   		objExcel.Cells(j+fila,10).Value = 1
   	End If
   Next
   
   'Lista de indices
   For i = 1 To 15 
   	objExcel.Cells(i+4,14).Value 	= listaIndices (i)
   	objExcel.Cells(i+4,16).Value 	= listaIndices (i+15)
   Next
   
   Dim NameInfDiario
   NameInfDiario = "C:\ESPACIO DE TRABAJO\InformeDiario\Pla" &(Replace(CStr(Date),"/","")& "-" &Replace(CStr(Time),":",""))&".xlsx"
   
   bfde4b54-0db7-4817-8032-87127bf19bb9 "Nombre del archivo: " & NameInfDiario
   objExcel.ActiveWorkbook.SaveAs NameInfDiario
   objExcel.ActiveWorkbook.Close
   objExcel.Application.Quit
   
   Set objExcel = Nothing
   	
   '#########################################################
   
   S07_InformeDiario_Planchas = NameInfDiario
   
   '888888888   GRABAR GATOS GRALES      8888888888
   
   Dim conngral, rstgral
   Dim hoy
   
   hoy = CStr(Year(DiaAnterior)) & "-" & CStr(Month(DiaAnterior)) & "-" & CStr(Day(DiaAnterior))
   
   Set conngral = CreateObject("ADODB.Connection")
   Set rstgral = CreateObject("ADODB.Recordset")
   
   'Open data source - Datenquelle öffnen
   conngral.Open "Provider=MSDASQL;Initial Catalog=Lavadero;DSN=Lavadero"
   'Error routine - Fehlerroutine
   If Err.Number <> 0 Then
   	bfde4b54-0db7-4817-8032-87127bf19bb9 "Conexion Error #" & Err.Number & " " & Err.Description
   	Err.Clear
   	conngral.close
   	Set conngral = Nothing  
   	Exit Function
   End If
   
   	SQL_Table = "INSERT INTO resultadosDiariosPlanchadoras VALUES ('"_
   		& DiaAnterior & "' , '" _
   		& Total2	(1) & "' , '" _
   		& Prod2		(1) & "' , '" _	
   		& Rend2		(1) & "' , '" _
   		& Total2	(2) & "' , '" _
   		& Prod2		(2) & "' , '" _
   		& Rend2		(2) & "' , '" _
   		& personas	(2) & "' , '" _
   		& Total2	(3) & "' , '" _
   		& Prod2		(3) & "' , '" _
   		& Rend2		(3) & "' , '" _
   		& personas	(3) & "' , '" _
   		& Total2	(4) & "' , '" _
   		& Prod2		(4) & "' , '" _
   		& Rend2		(4) & "' , '" _
   		& personas	(4) & "' , '" _
   		& Total2	(5) & "' , '" _
   		& Prod2		(5) & "' , '" _
   		& Rend2		(5) & "' , '" _
   		& personas	(5) & "')"
   
   	
   	Set rstgral = conngral.Execute(SQL_Table)
   
   	'Error routine
   	If Err.Number <> 0 Then
   		bfde4b54-0db7-4817-8032-87127bf19bb9 "Error Registrar datos GRales Planchas: #" & Err.Number & " " & Err.Description
   	End If
   	
   Err.Clear
   conngral.close
   Set conngral = Nothing
   Set rstgral = Nothing 

VB script "S100_LeerCliente"
   'Declaracion de Variables locales
   Dim conn, rst, SQL_Table
   
   On Error Resume Next
   
   Set conn = CreateObject("ADODB.Connection")
   Set rst = CreateObject("ADODB.Recordset")
   
   'Abrir BDD
   conn.Open "Provider=MSDASQL;Initial Catalog=Lavadero;DSN=Lavadero"
   
   
   'Chequeo de error
   If Err.Number <> 0 Then
   	bfde4b54-0db7-4817-8032-87127bf19bb9 "Error #" & Err.Number & " " & Err.Description
   	Err.Clear 
   	Set conn = Nothing
   	Exit Sub
   End If
   
   
   SQL_Table = "SELECT * FROM Cli_Lavadoras WHERE  ID = '" & SmartTags("Cli_ID") &"';"
   
   'Ejecutar consulta
   Set rst = conn.Execute(SQL_Table)
   
   SmartTags("Cli_Name") = rst.Fields(1).Value
   
   rst.close 
   
   conn.close
   
   Set rst = Nothing
   Set conn = Nothing

VB script "S101_EscribirCliente"
   'Declaracion de variables locales
   Dim conn, rst, SQL_Table, fechapl, fecha, hora
   
   On Error Resume Next
   
   Set conn = CreateObject("ADODB.Connection")
   Set rst = CreateObject("ADODB.Recordset")
   
   'Abrir BBDD
   conn.Open "Provider=MSDASQL;Initial Catalog=Lavadero;DSN=Lavadero"
   'conn.Open "Provider=MSDASQL;Initial Catalog=" & SmartTags("szDatabase") & ";DSN="&Database_Name&"" 'DSN= name of the odbc database - DSN= Name der ODBC-Datenbank
   
   'Crear consulta de insersion
   SQL_Table = "INSERT INTO Cli_Lavadoras VALUES ('"_
   		& SmartTags("ID_Nuevo")_
   		& "' , '" & SmartTags("Name_Nuevo") & "')"
   
   Set rst = conn.Execute(SQL_Table)
   
   'Error routine - Fehlerroutine
   If Err.Number <> 0 Then
   	bfde4b54-0db7-4817-8032-87127bf19bb9 "Error abrirb base #" & Err.Number & " " & Err.Description
   	Err.Clear
   	Set conn = Nothing 
   	Exit Sub
   End If
   
   conn.close
   
   Set rst = Nothing
   Set conn = Nothing

VB script "S102_CambiarCliente"
   'Declaracion de variables locales
   Dim conn, rst, SQL_Table
   
   On Error Resume Next
   
   Set conn = CreateObject("ADODB.Connection")
   Set rst = CreateObject("ADODB.Recordset")
   
   'Abrir BBDD
   conn.Open "Provider=MSDASQL;Initial Catalog=Lavadero;DSN=Lavadero"
   
   'Crear consulta de insersion
   SQL_Table = "UPDATE Cli_Lavadoras SET Empresa = '"_
   		& SmartTags("Name_Cambiar")_
   		& "' WHERE ID = '" & SmartTags("ID_Cambiar") & "';"
   
   Set rst = conn.Execute(SQL_Table)
   
   'Error routine - Fehlerroutine
   If Err.Number <> 0 Then
   	bfde4b54-0db7-4817-8032-87127bf19bb9 "Error abrirb base #" & Err.Number & " " & Err.Description
   	Err.Clear
   	Set conn = Nothing 
   	Exit Sub
   End If
   
   conn.close
   
   Set rst = Nothing
   Set conn = Nothing

VB script "S103_ActualizarLista"
   'Declaracion de Variables locales
   Dim conn, rst, SQL_Table
   
   On Error Resume Next
   
   Set conn = CreateObject("ADODB.Connection")
   Set rst = CreateObject("ADODB.Recordset")
   
   'Abrir BDD
   conn.Open "Provider=MSDASQL;Initial Catalog=Lavadero;DSN=Lavadero"
   
   
   'Chequeo de error
   If Err.Number <> 0 Then
   	bfde4b54-0db7-4817-8032-87127bf19bb9 "Error #" & Err.Number & " " & Err.Description
   	Err.Clear 
   	Set conn = Nothing
   	Exit Sub
   End If
   
   If (SmartTags("ID_1") <= 0) Then
   	SmartTags("ID_1") = 1
   End If
   
   SQL_Table = "SELECT * FROM Cli_Lavadoras WHERE  ID >= '" & SmartTags("ID_1") &"' ORDER BY ID;"
   
   'Ejecutar consulta
   Set rst = conn.Execute(SQL_Table)
   
   
   'Llenado de variables que muestan la lista
   If rst.EOF = False Then
   	SmartTags("ID_1") = rst.Fields(0).Value
   	SmartTags("Name_1") = rst.Fields(1).Value
   	rst.MoveNext
   Else
   	SmartTags("ID_1") = 0
   	SmartTags("Name_1") = "Vacio"
   End If
   
   If rst.EOF = False Then
   	SmartTags("ID_2") = rst.Fields(0).Value
   	SmartTags("Name_2") = rst.Fields(1).Value
   	rst.MoveNext
   Else
   	SmartTags("ID_2") = 0
   	SmartTags("Name_2") = "Vacio"
   End If
   
   If rst.EOF = False Then
   	SmartTags("ID_3") = rst.Fields(0).Value
   	SmartTags("Name_3") = rst.Fields(1).Value
   	rst.MoveNext
   Else
   	SmartTags("ID_3") = 0
   	SmartTags("Name_3") = "Vacio"
   End If
   
   If rst.EOF = False Then
   	SmartTags("ID_4") = rst.Fields(0).Value
   	SmartTags("Name_4") = rst.Fields(1).Value
   	rst.MoveNext
   Else
   	SmartTags("ID_4") = 0
   	SmartTags("Name_4") = "Vacio"
   End If
   
   If rst.EOF = False Then
   	SmartTags("ID_5") = rst.Fields(0).Value
   	SmartTags("Name_5") = rst.Fields(1).Value
   	rst.MoveNext
   Else
   	SmartTags("ID_5") = 0
   	SmartTags("Name_5") = "Vacio"
   End If
   
   
   rst.close
   
   conn.close
   
   Set rst = Nothing
   Set conn = Nothing

VB script "S200_CambSupervisor"
   'Declaracion de variables locales
   Dim conn, rst, SQL_Table
   
   On Error Resume Next
   
   Set conn = CreateObject("ADODB.Connection")
   Set rst = CreateObject("ADODB.Recordset")
   
   'Abrir BBDD
   conn.Open "Provider=MSDASQL;Initial Catalog=Lavadero;DSN=Lavadero"
   'conn.Open "Provider=MSDASQL;Initial Catalog=" & SmartTags("szDatabase") & ";DSN="&Database_Name&"" 'DSN= name of the odbc database - DSN= Name der ODBC-Datenbank
   
   
   
   'Crear consulta de insersion
   SQL_Table = "UPDATE Supervisores SET Supervisor = '"_
   		& SmartTags("Supervisor_Camb")_
   		& "' WHERE ID = '" & SmartTags("Supervisor_ID_Camb") & "';"
   
   Set rst = conn.Execute(SQL_Table)
   
   'Error routine - Fehlerroutine
   If Err.Number <> 0 Then
   	bfde4b54-0db7-4817-8032-87127bf19bb9 "Error abrirb base #" & Err.Number & " " & Err.Description
   	Err.Clear
   	Set conn = Nothing 
   	Exit Sub
   End If
   
   conn.close
   
   Set rst = Nothing
   Set conn = Nothing
   
   S201_ActualizarSupervisor()

VB script "S201_ActualizarSupervisor"
   'Declaracion de variables locales
   Dim conn, rst, SQL_Table
   
   On Error Resume Next
   
   Set conn = CreateObject("ADODB.Connection")
   Set rst = CreateObject("ADODB.Recordset")
   
   'Abrir BBDD
   conn.Open "Provider=MSDASQL;Initial Catalog=Lavadero;DSN=Lavadero"
   'conn.Open "Provider=MSDASQL;Initial Catalog=" & SmartTags("szDatabase") & ";DSN="&Database_Name&"" 'DSN= name of the odbc database - DSN= Name der ODBC-Datenbank
   
   
   SQL_Table = "SELECT * FROM Supervisores ORDER BY ID;"
   
   'Ejecutar consulta
   Set rst = conn.Execute(SQL_Table)
   
   
   'Llenado de variables que muestan la lista
   If rst.EOF = False Then
   	
   	SmartTags("Supervisor_Name_1") = rst.Fields(1).Value
   	rst.MoveNext
   
   	SmartTags("Supervisor_Name_2") = rst.Fields(1).Value
   	rst.MoveNext
   
   	SmartTags("Supervisor_Name_3") = rst.Fields(1).Value
   	rst.MoveNext
   
   	SmartTags("Supervisor_Name_4") = rst.Fields(1).Value
   
   End If
   
   conn.close
   
   Set rst = Nothing
   Set conn = Nothing

VB script "S15_Write_data_Lav2"
   On Error Resume Next
   Dim hayError, K
   hayError = False
   
   If SmartTags("Lav2_GrabarBDD") = True Then
   
   'Declaration of local tags
   Dim conn, rst, SQL_Table
   
   On Error Resume Next
   
   Set conn = CreateObject("ADODB.Connection")
   Set rst = CreateObject("ADODB.Recordset")
   
   'Abrir BBDD
   conn.Open "Provider=MSDASQL;Initial Catalog=Lavadero;DSN=Lavadero"
   
   'Error routine
   If Err.Number <> 0 Then
   	bfde4b54-0db7-4817-8032-87127bf19bb9 "Lav2: Error abrirb base #" & Err.Number & " " & Err.Description
   	hayError = True
   End If
   	
   	
   ' Recoleccion de datos de la lavadora 2
   Dim fechafin, fechainicio, cliente_0, cliente_1, cliente_2, operario, carga, programa, ciclovalido, falla, valido_CN
   
   
   
   'fecha actual
   fechafin = DateSerial(S12_Conversor_BCD_to_Int(SmartTags("Lav2_FchFin_Ano")), S12_Conversor_BCD_to_Int(SmartTags("Lav2_FchFin_Mes")), S12_Conversor_BCD_to_Int(SmartTags("Lav2_FchFin_Dia")))
   fechafin = fechafin + TimeSerial(S12_Conversor_BCD_to_Int(SmartTags("Lav2_FchFin_Hr")), S12_Conversor_BCD_to_Int(SmartTags("Lav2_FchFin_Min")), S12_Conversor_BCD_to_Int(SmartTags("Lav2_FchFin_Seg")))
   
   'fecha de inicio del ciclo
   fechainicio = DateSerial(S12_Conversor_BCD_to_Int(SmartTags("Lav2_FchIni_Ano")), S12_Conversor_BCD_to_Int(SmartTags("Lav2_FchIni_Mes")), S12_Conversor_BCD_to_Int(SmartTags("Lav2_FchIni_Dia")))
   fechainicio = fechainicio + TimeSerial(S12_Conversor_BCD_to_Int(SmartTags("Lav2_FchIni_Hr")), S12_Conversor_BCD_to_Int(SmartTags("Lav2_FchIni_Min")), S12_Conversor_BCD_to_Int(SmartTags("Lav2_FchIni_Seg")))
   
   cliente_0 = SmartTags("Lav2_Cliente_0")
   cliente_1 = SmartTags("Lav2_Cliente_1")
   cliente_2 = SmartTags("Lav2_Cliente_2")
   	
   operario = SmartTags("Lav2_Operador")
   
   carga = SmartTags("Lav2_CantRopa")
   
   programa = S12_Conversor_BCD_to_Int(SmartTags("Lav2_Programa"))
   
   falla = SmartTags("Lav2_Falla")
   
   	If SmartTags("Lav2_St_Ciclo") = 0 Then
   		valido_CN = 1
   	Else
   		valido_CN = 0
   	End If
   
   	If SmartTags("Lav2_St_Ciclo") = 0 Or  S12_Conversor_BCD_to_Int(SmartTags("Lav2_St_Ciclo")) > 13 Then	
   		ciclovalido = 1
   	Else
   		ciclovalido = 0
   	End If
   
   'Definition of data record - Definition des Datensatzes
   SQL_Table = "INSERT INTO Lav2 VALUES ('"_
   	& fechafin & "' , '" _
   	& fechainicio & "' , '" _
   	& cliente_0 & "' , '" _
   	& cliente_1 & "' , '" _
   	& cliente_2 & "' , '" _
   	& operario & "' , '" _
   	& carga & "' , '" _
   	& programa & "' , '" _
   	& ciclovalido & "' , '" _
   	& valido_CN & "')"
   	
   If hayError = False Then
   	'Execute - Ausführen
   	Set rst = conn.Execute(SQL_Table)
   End If
   
   	' Se guarda en lavado anterior
   	SmartTags("Lav2_Programa_Anterior") = SmartTags("Lav2_Programa")
   
   
   'Error routine - Fehler Routine
   If Err.Number <> 0 Then
   	bfde4b54-0db7-4817-8032-87127bf19bb9 "Error select Lav2: #" & Err.Number & " " & Err.Description
   	SmartTags("_errorNum2") = Err.Number
   	hayError = True
   End If
   
   	If hayError = False Or SmartTags("Lav2_Cont_IntentosGrabado") >= 3 Then
   		'Tres confirmaciones diferentes si es que no se proceso la anterior, con loops se tilda
   		If SmartTags("Lav2_GrabarBDD") = True Then
   			SmartTags("Lav2_Ciclograbado") = True
   		End If
   		K = Timer + 2
   		Do While (Timer<K)
   		Loop
   		If SmartTags("Lav2_GrabarBDD") = True Then
   			SmartTags("Lav2_Ciclograbado") = True
   		End If
   
   		
   				
   		If SmartTags("Lav2_Cont_IntentosGrabado") >= 3 Then
   			
   			'Envio email avisando que el ciclo no se grabo
   			cliente_0 = cliente_0 + cliente_1 + cliente_2
   			Call SA4_ErrorEnGrabBDD(2, fechafin, fechainicio, cliente_0,operario,carga,programa,ciclovalido)
   			
   			SmartTags("Lav2_Cont_IntentosGrabado") = 0
   			
   			If SmartTags("Lav2_GrabarBDD") = True Then
   				SmartTags("Lav2_Ciclograbado") = True
   			End If	
   		
   		End If
   		
   	Else
   			
   		SmartTags("Lav2_Cont_IntentosGrabado") = SmartTags("Lav2_Cont_IntentosGrabado") + 1
   		
   	End If
   
   
   
   
   End If
   	
   ' Jump de error en esta linea
   	
   Err.Clear
   'Close data source 
   conn.close
   Set conn = Nothing
   Set rst = Nothing 
   	

VB script "S16_Write_data_Lav3"
   On Error Resume Next
   Dim hayError, K
   hayError = False
   
   If SmartTags("Lav3_GrabarBDD") = True Then
   
   'Declaration of local tags
   Dim conn, rst, SQL_Table
   
   Set conn = CreateObject("ADODB.Connection")
   Set rst = CreateObject("ADODB.Recordset")
   
   'Abrir BBDD
   conn.Open "Provider=MSDASQL;Initial Catalog=Lavadero;DSN=Lavadero"
   
   'Error routine - Fehlerroutine
   If Err.Number <> 0 Then
   	bfde4b54-0db7-4817-8032-87127bf19bb9 "Lav3: Error abrirb base #" & Err.Number & " " & Err.Description
   	hayError = True
   End If
   	
   	
   ' Recoleccion de datos de la lavadora 3 
   Dim fechafin, fechainicio, cliente_0, cliente_1, cliente_2, operario, carga, programa, ciclovalido, falla, valido_CN
   
   'fecha actual
   fechafin = DateSerial(S12_Conversor_BCD_to_Int(SmartTags("Lav3_FchFin_Ano")), S12_Conversor_BCD_to_Int(SmartTags("Lav3_FchFin_Mes")), S12_Conversor_BCD_to_Int(SmartTags("Lav3_FchFin_Dia")))
   'fechafin = DateSerial(S12_Conversor_BCD_to_Int(SmartTags("Lav3_FchFin_Ano")), S12_Conversor_BCD_to_Int(SmartTags("Lav3_FchFin_Mes")), Day(Date()))
   fechafin = fechafin + TimeSerial(S12_Conversor_BCD_to_Int(SmartTags("Lav3_FchFin_Hr")), S12_Conversor_BCD_to_Int(SmartTags("Lav3_FchFin_Min")), S12_Conversor_BCD_to_Int(SmartTags("Lav3_FchFin_Seg")))
   
   'fecha de inicio del ciclo
   fechainicio = DateSerial(S12_Conversor_BCD_to_Int(SmartTags("Lav3_FchIni_Ano")), S12_Conversor_BCD_to_Int(SmartTags("Lav3_FchIni_Mes")), S12_Conversor_BCD_to_Int(SmartTags("Lav3_FchIni_Dia")))
   fechainicio = fechainicio + TimeSerial(S12_Conversor_BCD_to_Int(SmartTags("Lav3_FchIni_Hr")), S12_Conversor_BCD_to_Int(SmartTags("Lav3_FchIni_Min")), S12_Conversor_BCD_to_Int(SmartTags("Lav3_FchIni_Seg")))
   
   cliente_0 = SmartTags("Lav3_Cliente_0")
   cliente_1 = SmartTags("Lav3_Cliente_1")
   cliente_2 = SmartTags("Lav3_Cliente_2")
   	
   operario = SmartTags("Lav3_Operador")
   
   carga = SmartTags("Lav3_CantRopa")
   
   programa = S12_Conversor_BCD_to_Int(SmartTags("Lav3_Programa"))
   
   falla = SmartTags("Lav3_Falla")
   
   	If SmartTags("Lav3_St_Ciclo") = 0 Then
   		valido_CN = 1
   	Else
   		valido_CN = 0
   	End If
   
   	If SmartTags("Lav3_St_Ciclo") = 0 Or  S12_Conversor_BCD_to_Int(SmartTags("Lav3_St_Ciclo")) > 13 Then	
   		ciclovalido = 1
   	Else
   		ciclovalido = 0
   	End If
   
   
   'Definition of data record - Definition des Datensatzes
   SQL_Table = "INSERT INTO Lav3 VALUES ('"_
   	& fechafin 		& "' , '" _
   	& fechainicio 	& "' , '" _
   	& cliente_0 	& "' , '" _
   	& cliente_1 	& "' , '" _
   	& cliente_2 	& "' , '" _
   	& operario 		& "' , '" _
   	& carga 		& "' , '" _
   	& programa 		& "' , '" _
   	& ciclovalido & "' , '" _
   	& valido_CN & "')"
   
   If hayError = False Then
   	'Execute - Ausführen
   	Set rst = conn.Execute(SQL_Table)
   End If
   
   'Se registra el ciclo anterior
   SmartTags("Lav3_Programa_Anterior") = SmartTags("Lav3_Programa")
   
   'Error routine - Fehler Routine
   If Err.Number <> 0 Then
   	bfde4b54-0db7-4817-8032-87127bf19bb9 "Error select Lav3: #" & Err.Number & " " & Err.Description
   	SmartTags("_errorNum3") = Err.Number
   	hayError = True
   End If
   
   
   	If hayError = False Or SmartTags("Lav3_Cont_IntentosGrabado") >= 3 Then
   		'Tres confirmaciones diferentes si es que no se proceso la anterior, con loops se tilda
   		If SmartTags("Lav3_GrabarBDD") = True Then
   			SmartTags("Lav3_Ciclograbado") = True
   		End If
   		K = Timer + 2
   		Do While (Timer<K)
   		Loop
   		If SmartTags("Lav3_GrabarBDD") = True Then
   			SmartTags("Lav3_Ciclograbado") = True
   		End If
   
   		If SmartTags("Lav3_Cont_IntentosGrabado") >= 3 Then
   			
   			'Envio email avisando que el ciclo no se grabo
   			cliente_0 = cliente_0 + cliente_1 + cliente_2
   			Call SA4_ErrorEnGrabBDD(3, fechafin, fechainicio, cliente_0,operario,carga,programa,ciclovalido)
   			
   			SmartTags("Lav3_Cont_IntentosGrabado") = 0
   			
   			If SmartTags("Lav3_GrabarBDD") = True Then
   				SmartTags("Lav3_Ciclograbado") = True
   			End If	
   		
   		End If
   		
   	Else
   			
   		SmartTags("Lav3_Cont_IntentosGrabado") = SmartTags("Lav3_Cont_IntentosGrabado") + 1
   		
   	End If
   
   End If
   
   ' Jump de error en esta linea
   
   Err.Clear
   'Close data source 
   conn.close
   Set conn = Nothing
   Set rst = Nothing 
   	
   	

VB script "S202_ActualizarSup_HMI"
   If 		SmartTags("Planchadora1_Supervisores{1}_Estado") = True Then
   	SmartTags("Supervisor_Name_Ahora") = SmartTags("Supervisor_Name_1")
   End If
   	
   If SmartTags("Planchadora1_Supervisores{2}_Estado") = True Then
   	SmartTags("Supervisor_Name_Ahora") = SmartTags("Supervisor_Name_2")
   End If
   
   If SmartTags("Planchadora1_Supervisores{3}_Estado") = True Then
   	SmartTags("Supervisor_Name_Ahora") = SmartTags("Supervisor_Name_3")
   End If
   
   If SmartTags("Planchadora1_Supervisores{4}_Estado") = True Then
   	SmartTags("Supervisor_Name_Ahora") = SmartTags("Supervisor_Name_4")
   End If
   
   If 		 (SmartTags("Planchadora1_Supervisores{1}_Estado") = False)_
   	 And (SmartTags("Planchadora1_Supervisores{2}_Estado") = False)_
   	 And (SmartTags("Planchadora1_Supervisores{3}_Estado") = False)_
   	 And (SmartTags("Planchadora1_Supervisores{4}_Estado") = False) Then
   			SmartTags("Supervisor_Name_Ahora") = "Nobody"
   End If

VB script "Prueba"
   'Informe de planchadoras
   bfde4b54-0db7-4817-8032-87127bf19bb9 "Se llamo a S07"
   Call S07_InformeDiario_Planchas()
   bfde4b54-0db7-4817-8032-87127bf19bb9 "Se Salio de S07"
   
   
   'Dim thoras, dias
   'thoras = FormatDateTime("2020-06-01 13:30:00", 4)
   'dias = 1
   'SmartTags("BCDtoInt")= SA2_TotalTimeToString(dias, thoras)
   
   ''SmartTags("Prueba_String") = "SELECT * FROM Lav1 WHERE cast(Fecha As Date) = '"_
   ''	& CStr(Year(Date)) & "-" & CStr(Month(Date)) & "-" & CStr(Day(Date)) & "' "_
   ''	& "AND cast(Fecha as time) >= '00:00:00' AND cast(Fecha as time) <= '23:50:00' order by Fecha"
   '
   'Dim final, inicial, salida, tiempodeprod, salida2
   '
   'final 	= FormatDateTime(CStr(SmartTags("date_prueba_f")), 4)
   'inicial	= FormatDateTime(CStr(SmartTags("date_prueba_i")), 4)
   '
   'tiempodeprod = FormatDateTime(CStr(SmartTags("date_prueba_prod")), 4)
   '
   'If Err.Number <> 0 Then
   '	ShowSystemAlarm "Error en prueba 1#" & Err.Number & " " & Err.Description
   '	Err.Clear
   '	Exit Sub
   'End If
   ' 
   '	salida = DateAdd("n",Minute(final) - Minute(inicial), salida)
   '	salida = DateAdd("h",Hour(final) - Hour(inicial), salida)
   '
   '	salida2 = DateAdd("n",Minute(salida) - Minute(tiempodeprod), salida2)
   '	salida2 = DateAdd("h",Hour(salida) - Hour(tiempodeprod), salida2)
   '	
   ''	If Second(tiempodeprod) <> 0 Then 
   ''		salida = DateAdd("s",Second(salida) - Second(tiempodeprod), salida)
   ''	End If
   ''	
   ''	If Minute(tiempodeprod) <> 0 Then
   ''		If Second(tiempodeprod) <> 0 Then
   ''			salida = DateAdd("n",Minute(salida) - Minute(tiempodeprod), salida)
   ''		Else
   ''			salida = DateAdd("n",Minute(salida) - Minute(tiempodeprod), salida)
   ''		End If
   ''	End If
   ''	
   ''	If Hour(tiempodeprod) <> 0 Then
   ''		If Minute(tiempodeprod) <> 0 Then
   ''			salida = DateAdd("h",Hour(salida) - Hour(tiempodeprod), salida)
   ''		Else
   ''			salida = DateAdd("h",Hour(salida) - Hour(tiempodeprod), salida)
   ''		End If
   ''	End If	
   '	
   '	
   'If Err.Number <> 0 Then
   '	ShowSystemAlarm "Error en prueba 2#" & Err.Number & " " & Err.Description
   '	Err.Clear
   '	Exit Sub
   'End If
   '	
   'SmartTags("date_prueba_o") = FormatDateTime(salida2, 4)
   '
   '
   'If Err.Number <> 0 Then
   '	ShowSystemAlarm "Error en prueba 3#" & Err.Number & " " & Err.Description
   '	Err.Clear
   '	Exit Sub
   'End If
   '	If Second(thorasSdate(i)) <> 0 Then 
   '		TiempoMuertoS(i) = DateAdd("s",60 - Second(thorasSdate(i)), TiempoMuertoS(i))
   '	End If
   '	
   '	If Minute(thorasdate) <> 0 Then
   '		If Second(thorasdate) <> 0 Then
   '			thorasmuertodate = DateAdd("n",59 - Minute(thorasdate), thorasmuertodate)
   '		Else
   '			thorasmuertodate = DateAdd("n",60 - Minute(thorasdate), thorasmuertodate)
   '		End If
   '	End If
   '	
   '	If Hour(thorasdate) <> 0 Then
   '		If Minute(thorasdate) <> 0 Then
   '			thorasmuertodate = DateAdd("h",23 - Hour(thorasdate), thorasmuertodate)
   '		Else
   '			thorasmuertodate = DateAdd("h",24 - Hour(thorasdate), thorasmuertodate)
   '		End If
   '	End If
   '	
   '	If Hour(thorasdate) = 0 And Minute(thorasdate) = 0 And Second(thorasdate) = 0 Then
   '		thorasmuertodate = DateAdd("h",24, thorasmuertodate)
   '	End If	
   	
   'Next

VB script "S300_LeerOperador"
   'Declaracion de Variables locales
   Dim conn21, rst21, SQL_Table
   
   On Error Resume Next
   
   Set conn21 = CreateObject("ADODB.Connection")
   Set rst21 = CreateObject("ADODB.Recordset")
   
   'Abrir BDD
   conn21.Open "Provider=MSDASQL;Initial Catalog=Lavadero;DSN=Lavadero"
   
   
   'Chequeo de error
   If Err.Number <> 0 Then
   	bfde4b54-0db7-4817-8032-87127bf19bb9 "Error #" & Err.Number & " " & Err.Description
   	Err.Clear 
   	Set conn21 = Nothing
   	Exit Sub
   End If
   
   SQL_Table = "SELECT * FROM Op_Lavadoras WHERE  ID = '" & SmartTags("OP_ID") &"';"
   
   'Ejecutar consulta
   Set rst21 = conn21.Execute(SQL_Table)
   
   SmartTags("OP_Name") = rst21.Fields(1).Value
   
   rst21.close 
   
   conn21.close
   
   Set rst21 = Nothing
   Set conn21 = Nothing

VB script "S301_EscribirOperador"
   'Declaracion de variables locales
   Dim conn301, rst301, SQL_Table, fechapl, fecha, hora
   
   On Error Resume Next
   
   Set conn301 = CreateObject("ADODB.Connection")
   Set rst301 = CreateObject("ADODB.Recordset")
   
   'Abrir BBDD
   conn301.Open "Provider=MSDASQL;Initial Catalog=Lavadero;DSN=Lavadero"
   'conn.Open "Provider=MSDASQL;Initial Catalog=" & SmartTags("szDatabase") & ";DSN="&Database_Name&"" 'DSN= name of the odbc database - DSN= Name der ODBC-Datenbank
   
   'Crear consulta de insersion
   SQL_Table = "INSERT INTO Op_Lavadoras VALUES ('"_
   		& SmartTags("ID_OP_Nuevo")_
   		& "' , '" & SmartTags("Name_OP_Nuevo") & "')"
   
   Set rst301 = conn301.Execute(SQL_Table)
   
   'Error routine - Fehlerroutine
   If Err.Number <> 0 Then
   	bfde4b54-0db7-4817-8032-87127bf19bb9 "Error abrirb base #" & Err.Number & " " & Err.Description
   	Err.Clear
   	Set conn301 = Nothing 
   	Exit Sub
   End If
   
   conn301.close
   
   Set rst301 = Nothing
   Set conn301 = Nothing

VB script "S302_CambiarOperador"
   'Declaracion de variables locales
   Dim conn302, rst302, SQL_Table
   
   On Error Resume Next
   
   Set conn302 = CreateObject("ADODB.Connection")
   Set rst302 = CreateObject("ADODB.Recordset")
   
   'Abrir BBDD
   conn302.Open "Provider=MSDASQL;Initial Catalog=Lavadero;DSN=Lavadero"
   'conn.Open "Provider=MSDASQL;Initial Catalog=" & SmartTags("szDatabase") & ";DSN="&Database_Name&"" 'DSN= name of the odbc database - DSN= Name der ODBC-Datenbank
   
   'Crear consulta de insersion
   SQL_Table = "UPDATE Op_Lavadoras SET Nombre = '"_
   		& SmartTags("Name_OP_Cambiar")_
   		& "' WHERE ID = '" & SmartTags("ID_OP_Cambiar") & "';"
   
   Set rst302 = conn302.Execute(SQL_Table)
   
   'Error routine - Fehlerroutine
   If Err.Number <> 0 Then
   	bfde4b54-0db7-4817-8032-87127bf19bb9 "Error abrirb base #" & Err.Number & " " & Err.Description
   	Err.Clear
   	Set conn302 = Nothing 
   	Exit Sub
   End If
   
   conn302.close
   
   Set rst302 = Nothing
   Set conn302 = Nothing

VB script "S303_ActualizarListaOp"
   'Declaracion de Variables locales
   Dim conn303, rst303, SQL_Table
   
   On Error Resume Next
   
   Set conn303 = CreateObject("ADODB.Connection")
   Set rst303 = CreateObject("ADODB.Recordset")
   
   'Abrir BDD
   conn303.Open "Provider=MSDASQL;Initial Catalog=Lavadero;DSN=Lavadero"
   
   
   'Chequeo de error
   If Err.Number <> 0 Then
   	bfde4b54-0db7-4817-8032-87127bf19bb9 "Error #" & Err.Number & " " & Err.Description
   	Err.Clear 
   	Set conn303 = Nothing
   	Exit Sub
   End If
   
   If (SmartTags("ID_OP_1") <= 0) Then
   	SmartTags("ID_OP_1") = 1
   End If
   
   SQL_Table = "SELECT * FROM Op_Lavadoras WHERE  ID >= '" & SmartTags("ID_OP_1") &"' ORDER BY ID;"
   
   'Ejecutar consulta
   Set rst303 = conn303.Execute(SQL_Table)
   
   
   'Llenado de variables que muestan la lista
   If rst303.EOF = False Then
   	SmartTags("ID_OP_1") = rst303.Fields(0).Value
   	SmartTags("Name_OP_1") = rst303.Fields(1).Value
   	rst303.MoveNext
   Else
   	SmartTags("ID_OP_1") = 0
   	SmartTags("Name_OP_1") = "Vacio"
   End If
   
   If rst303.EOF = False Then
   	SmartTags("ID_OP_2") = rst303.Fields(0).Value
   	SmartTags("Name_OP_2") = rst303.Fields(1).Value
   	rst303.MoveNext
   Else
   	SmartTags("ID_OP_2") = 0
   	SmartTags("Name_OP_2") = "Vacio"
   End If
   
   If rst303.EOF = False Then
   	SmartTags("ID_OP_3") = rst303.Fields(0).Value
   	SmartTags("Name_OP_3") = rst303.Fields(1).Value
   	rst303.MoveNext
   Else
   	SmartTags("ID_OP_3") = 0
   	SmartTags("Name_OP_3") = "Vacio"
   End If
   
